// TwinCAT 3 PLC project CP_5C7432
// libraries:
//   AutomationBaseClasses, * (PTW TU Darmstadt)
//   Tc2_ControllerToolbox, * (Beckhoff Automation GmbH)
//   Tc2_Coupler, * (Beckhoff Automation GmbH)
//   Tc2_DALI, * (Beckhoff Automation GmbH)
//   Tc2_EIB, * (Beckhoff Automation GmbH)
//   Tc2_EtherCAT, * (Beckhoff Automation GmbH)
//   Tc2_IoFunctions, * (Beckhoff Automation GmbH)
//   Tc2_LON, * (Beckhoff Automation GmbH)
//   Tc2_MBus, * (Beckhoff Automation GmbH)
//   Tc2_ModbusRTU, * (Beckhoff Automation GmbH)
//   Tc2_ModbusSrv, * (Beckhoff Automation GmbH)
//   Tc2_Standard, * (Beckhoff Automation GmbH)
//   Tc2_Standard, * (Beckhoff Automation GmbH)
//   Tc2_System, * (Beckhoff Automation GmbH)
//   Tc2_System, * (Beckhoff Automation GmbH)
//   Tc2_SystemCX, * (Beckhoff Automation GmbH)
//   Tc2_Utilities, * (Beckhoff Automation GmbH)
//   Tc3_Module, * (Beckhoff Automation GmbH)
//   Tc3_Module, * (Beckhoff Automation GmbH)
//   Tc3_PLCopen_OpcUa, * (Beckhoff Automation GmbH)
// project tree:
//   DUTs/01 Actuators/pcmChiller/ E_PCMControlMode.TcDUT, ST_pcmChillerDefaultParameters.TcDUT, ST_pcmChillerState.TcDUT
//   DUTs/02 Sensors/ ST_JanitzaState.TcDUT
//   DUTs/03 Storages/BufferStorage/ ST_BufferStorageState.TcDUT
//   DUTs/03 Storages/HVFAStorage/ ST_HVFAStorageState.TcDUT (not stored), ST_HVFAStorageSystemDefaultParameters.TcDUT (not stored)
//   DUTs/03 Storages/PCMStorage/ ST_PCMStorageState.TcDUT
//   DUTs/03 Storages/VSIStorage/ ST_VSIStorageState.TcDUT (not stored), ST_VSIStorageSystemDefaultParameters.TcDUT (not stored)
//   DUTs/04 Systems/ConsumerSystems/CN/ ST_CN_CentralMachineCoolingDefaultParameters.TcDUT, ST_FlywheelMassStorageDefaultParameters.TcDUT
//   DUTs/04 Systems/ConsumerSystems/HNHT/ ST_AnnealingOvenExhaustGasDefaultParameters.TcDUT, ST_HNHT_CentralMachineHeatingDefaultParameters.TcDUT, ST_StaticHeatingDefaultParameters.TcDUT (not stored)
//   DUTs/04 Systems/ConsumerSystems/HNLT/ ST_AnnealingOvenSealingDefaultParameters.TcDUT (not stored), ST_DCSystemDefaultParameters.TcDUT, ST_CompressorDefaultParameters.TcDUT (not stored)
//   DUTs/04 Systems/CoolingSystems/AbsorptionChillerSystem/ ST_AbsorptionChillerDefaultParameters.TcDUT (not stored)
//   DUTs/04 Systems/CoolingSystems/eChiller/ ST_eChillerDefaultParameters.TcDUT, ST_eChillerState.TcDUT
//   DUTs/04 Systems/CoolingSystems/OuterCapillaryTubeMats/ ST_OuterCapillaryTubeMatsDefaultParameters.TcDUT (not stored)
//   DUTs/04 Systems/HeatingSystems/CHP/ E_CHPControlMode.TcDUT, ST_CHPDefaultParameters.TcDUT, ST_CHPSetParameters.TcDUT, ST_CHPState.TcDUT
//   DUTs/04 Systems/HeatingSystems/CondensingBoiler/ ST_CondensingBoilerDefaultParameters.TcDUT, ST_CondensingBoilerState.TcDUT
//   DUTs/04 Systems/HeatingSystems/HeatPump/ ST_HeatPumpDefaultParameters.TcDUT, ST_HeatPumpState.TcDUT
//   DUTs/04 Systems/LinkageSystems/HeatExchanger1/ ST_HeatExchanger1DefaultParameters.TcDUT
//   DUTs/04 Systems/LinkageSystems/InnerCapillaryTubeMats/ ST_InnerCapillaryTubeMatsDefaultParameters.TcDUT, ST_InnerCapillaryTubeMatsSetParameters.TcDUT (not stored)
//   DUTs/04 Systems/LinkageSystems/PCMSystem/ E_PCMSystemControlMode.TcDUT, ST_PCMSystemSetParameters.TcDUT
//   DUTs/04 Systems/LinkageSystems/UnderfloorHeating/ ST_UnderfloorHeatingDefaultParameters.TcDUT (not stored), ST_UnderfloorHeatingSetParameters.TcDUT (not stored)
//   DUTs/04 Systems/LinkageSystems/Ventilation/ ST_VentilationDefaultParameters.TcDUT, ST_VentilationSetParameters.TcDUT, ST_VentilationState.TcDUT
//   DUTs/04 Systems/StorageSystems/ ST_ActiveStorageSystemSetParameters.TcDUT (not stored), ST_ActiveStorageSystemState.TcDUT
//   DUTs/05 Thermal Networks/ ST_AmbientState.TcDUT, ST_CoolingNetworkControl.TcDUT, ST_HeatingNetworkHighTemperatureControl.TcDUT, ST_HnhtHnltLinkageControl.TcDUT, ST_HnltCnLinkageControl.TcDUT (not stored), ST_HeatingNetworkLowTemperatureControl.TcDUT (not stored), ST_HnhtCnLinkageControl.TcDUT, ST_ThermalNetworkState.TcDUT (not stored)
//   DUTs/06 Strategy/ ST_StrategyDefaultParameters.TcDUT, ST_StrategySetParameters.TcDUT, ST_StrategyState.TcDUT
//   DUTs/07 Utilities/ ST_OPC_UANode.TcDUT, ST_OPC_UA_Server.TcDUT (not stored)
//   DUTs/08 Lighting/Einzelanlagen/Beleuchtung %28Bel%29/ ST_Bel_Lampen_Monitoring.TcDUT (not stored), ST_Bel_Parameter.TcDUT (not stored), ST_Bel_RGBW_Steuerung.TcDUT (not stored), ST_Bel_RGBW_Zustand.TcDUT (not stored), ST_Bel_Stellwert.TcDUT (not stored), ST_Bel_Steuerung.TcDUT (not stored), ST_Bel_Zustand.TcDUT (not stored)
//   DUTs/08 Lighting/Einzelanlagen/RGBW-Kanal/ ST_RGBW_Steuerung.TcDUT (not stored), ST_RGBW_Zustand.TcDUT (not stored)
//   DUTs/08 Lighting/Library/Allgemein/ ST_Steuerung_auto_manu_BOOL.TcDUT (not stored), ST_Steuerung_auto_manu_opti_BOOL.TcDUT (not stored), ST_Steuerung_auto_manu_opti_REAL.TcDUT (not stored), ST_Steuerung_auto_manu_opti_SINT.TcDUT (not stored), ST_Steuerung_auto_manu_String.TcDUT (not stored), ST_Zustand_Netze_Anford.TcDUT (not stored), ST_Zustand_Netz_Anford.TcDUT (not stored)
//   DUTs/08 Lighting/Sonstige/ ST_GA_global.TcDUT (not stored), ST_Initialisierungsroutine.TcDUT (not stored)
//   DUTs/08 Lighting/Systeme/Beleuchtung %28Bel%29/ ST_System_Bel_Parameter.TcDUT (not stored), ST_System_Bel_Stellwert.TcDUT (not stored), ST_System_Bel_Steuerung.TcDUT (not stored), ST_System_Bel_Zustand.TcDUT (not stored)
//   GVLs/ GlobalVariables.TcGVL, M_Bus.TcGVL
//   GVLs/Lighting %28from old implementation%29/ Con_Bel.TcGVL (not stored), Global_Variables.TcGVL (not stored), Variablen_Konfiguration.TcGVL (not stored)
//   / MBus_WZaehler_Task.TcTTO, MBus_Zaehler_Task.TcTTO, Standard.TcTTO
//   POUs/01 Actuators/ConsumerUnits/ FB_AnnealingOven.TcPOU, FB_EMAG_GT.TcPOU, FB_DC.TcPOU, FB_EMAG_Y.TcPOU, FB_MAFAC_Java.TcPOU, FB_FlywheelMassStorage.TcPOU, FB_BvL_CleaningSystem.TcPOU, FB_Ventilation.TcPOU
//   POUs/01 Actuators/CoolingUnits/ FB_eChiller.TcPOU, FB_PCMChiller.TcPOU
//   POUs/01 Actuators/HeatingUnits/ FB_CHP.TcPOU, FB_HeatPump.TcPOU, FB_CondensingBoiler.TcPOU
//   POUs/01 Actuators/Pumps/ FB_Pump2Point.TcPOU
//   POUs/02 Sensors/ FB_JanitzaSensor.TcPOU, FB_LowVoltageMainDistribution.TcPOU, FB_WeatherStation.TcPOU
//   POUs/03 Storages/ FB_BufferStorage.TcPOU, FB_PCMStorage.TcPOU, FB_VSIStorage.TcPOU, FB_HVFAStorage.TcPOU
//   POUs/04 Systems/ConsumerSystems/CN/ FB_CN_CentralMachineCooling.TcPOU, FB_FlywheelMassStorageSystem.TcPOU
//   POUs/04 Systems/ConsumerSystems/HNHT/ FB_AnnealingOvenExhaustGasSystem.TcPOU, FB_HNHT_CentralMachineHeating.TcPOU, FB_StaticHeatingSystem.TcPOU
//   POUs/04 Systems/ConsumerSystems/HNLT/ FB_AnnealingOvenSealingSystem.TcPOU, FB_DCSystem.TcPOU, FB_CompressorSystem.TcPOU
//   POUs/04 Systems/CoolingSystems/ FB_AbsorptionChillerSystem.TcPOU, FB_eChillerSystem.TcPOU, FB_OuterCapillaryTubeMats.TcPOU, FB_PCMSupplySystem.TcPOU
//   POUs/04 Systems/HeatingSystems/ FB_CHPSystem.TcPOU, FB_CondensingBoilerSystem.TcPOU
//   POUs/04 Systems/LinkageSystems/ FB_HeatExchanger1System.TcPOU, FB_HeatPumpSystem_CN.TcPOU, FB_HeatPumpSystem_HNHT.TcPOU, FB_InnerCapillaryTubeMats.TcPOU, FB_UnderfloorHeatingSystem.TcPOU, FB_VentilationSystem.TcPOU
//   POUs/04 Systems/StorageSystems/ FB_HVFAStorageSystem.TcPOU, FB_VSIStorageSystem.TcPOU
//   POUs/05 Thermal Networks/ FB_Ambient.TcPOU, FB_CoolingNetwork.TcPOU, FB_HeatingNetworkHighTemperature.TcPOU, FB_HnhtCnLinkage.TcPOU, FB_HnhtHnltLinkage.TcPOU, FB_HnltCnLinkage.TcPOU, FB_HeatingNetworkLowTemperature.TcPOU
//   POUs/06 Strategy/ FB_StrategyController.TcPOU, FB_StrategyController_noChiller.TcPOU, FB_StrategyController_NoStorages.TcPOU, FB_StrategyController_Conventional.TcPOU
//   POUs/07 Utilities/ FB_OPC_UA_Read.TcPOU
//   POUs/08 Lighting/Einzelanlagen/Beleuchtung %28Bel%29/Bel_RGBW/ FB_Bel_Einzel_farbe.TcPOU (not stored), FB_Bel_Einzel_farbe_1.TcPOU (not stored), FB_Bel_RGBW.TcPOU (not stored), FB_Bel_RGBW_Ablaufsteuerung.TcPOU (not stored), FB_Bel_RGBW_Logik.TcPOU (not stored), FB_Bel_RGBW_Regelung.TcPOU (not stored), FB_Bel_RGBW_Sued.TcPOU (not stored) (excluded from build)
//   POUs/08 Lighting/Einzelanlagen/Beleuchtung %28Bel%29/ FB_Bel.TcPOU (not stored), FB_Bel_Ablaufsteuerung.TcPOU (not stored), FB_Bel_Filter.TcPOU (not stored), FB_Bel_Input.TcPOU (not stored), FB_Bel_Lichtsensor.TcPOU (not stored), FB_Bel_Logik.TcPOU (not stored), FB_Bel_Monitoring.TcPOU (not stored), FB_Bel_Output.TcPOU (not stored), FB_Bel_Sollwertscheck.TcPOU (not stored), FB_Bel_Stellwertscheck.TcPOU (not stored), FB_Bel_Steuerung.TcPOU (not stored), FB_Bel_Taster.TcPOU (not stored), FB_Bel_Taster_Steuerung.TcPOU (not stored), FB_Bel_Zustandscheck.TcPOU (not stored), F_Bel_Daten_Lesen.TcPOU (not stored), F_Bel_Daten_Schreiben.TcPOU (not stored)
//   POUs/08 Lighting/ FB_GA_Allgemein.TcPOU, FB_Initialisierungsroutine.TcPOU
//   POUs/08 Lighting/Library %28allgemein%29/ FB_SetResetFallTrigger.TcPOU (not stored)
//   POUs/08 Lighting/Systeme/Sonstiges/Beleuchtung/Beleuchtung Außen/ FB_System_BelAu.TcPOU (not stored), FB_System_BelAu_Ablaufsteuerung.TcPOU (not stored), FB_System_BelAu_Logik.TcPOU, FB_System_BelAu_Regelung.TcPOU, FB_System_BelAu_Sensorik.TcPOU, FB_System_BelAu_Sollwertscheck.TcPOU (not stored), FB_System_BelAu_Stellwertscheck.TcPOU (not stored), FB_System_BelAu_Zustandscheck.TcPOU (not stored)
//   POUs/08 Lighting/Systeme/Sonstiges/Beleuchtung/Beleuchtung Halle/ FB_System_BelHa.TcPOU (not stored), FB_System_BelHa_Ablaufsteuerung.TcPOU, FB_System_BelHa_Logik.TcPOU (not stored), FB_System_BelHa_Regelung.TcPOU (not stored), FB_System_BelHa_Sensorik.TcPOU, FB_System_BelHa_Sollwertscheck.TcPOU (not stored), FB_System_BelHa_Stellwertscheck.TcPOU, FB_System_BelHa_Zustandscheck.TcPOU
//   POUs/08 Lighting/Systeme/Sonstiges/Beleuchtung/ FB_Beleuchtung.TcPOU, FB_System_Bel_Zustandscheck.TcPOU (not stored)
//   POUs/ MAIN.TcPOU, MBUS_WZaehler.TcPOU, MBUS_WZaehler2.TcPOU, MBUS_WZaehler_Basement.TcPOU, MBUS_Zaehler.TcPOU
// real-time tasks:
//   TASK MBus_Zaehler_Task: cycle T#10ms, priority 8, ADS port 351
//   TASK Standard: cycle T#20ms, priority 10, ADS port 352
//   TASK MBus_WZaehler_Task: cycle T#6ms, priority 6, ADS port 353
//   TASK Gerät 7 (OPC UA Virtual)_Task_58: cycle T#40ms, priority 12, ADS port 350
// I/O:
//   DEVICE Gerät 6 (EL6731), AmsNetId 0.0.0.0.7.1
//     Box 1 (CIM/CIU 150 pump) // Vendor: GRUNDFOS Revision: R1 PU361
//     Box 2 (CIM/CIU 150 pump) // Vendor: GRUNDFOS Revision: R1 PU261
//     Box 3 (CIM/CIU 150 pump) // Vendor: GRUNDFOS Revision: R1 PU300
//     Box 4 (CIM/CIU 150 pump) // Vendor: GRUNDFOS Revision: R1 PU100
//     Box 5 (CIM/CIU 150 pump) // Vendor: GRUNDFOS Revision: R1 PU145
//     Box 6 (CIM/CIU 150 pump) // Vendor: GRUNDFOS Revision: R1 PU245
//   DEVICE Gerät 10 (EtherCAT), AmsNetId 0.0.0.0.11.1
//     Term 31 (EK1100) [EK1100 EtherCAT Coupler (2A E-Bus)]
//       Term 30 (EL6070-0033) [EL6070-0033 1Ch. Licence key terminal, individual licences]
//       Profibus_1 (EL6731) [EL6731 PROFIBUS DP Master]
//       Profibus_2 (EL6731) [EL6731 PROFIBUS DP Master]
//       Box 3 (BK1250)
//     Klemme 15 (EK1100) [EK1100 EtherCAT-Koppler (2A E-Bus)]
//       Klemme 27 (EL3068) [EL3068 8K. Ana. Eingang 0-10V]
//       Klemme 28 (EL4008) [EL4008 8K. Ana. Ausgang 0-10V, 12bit]
//       Klemme 39 (EK1521-0010) [EK1521-0010 1-Port EtherCAT-Abzweig (FX-SingleMode)]
//         Klemme 40 (EK1501-0010) [EK1501-0010 EtherCAT-Koppler (2A E-Bus, FX-SingleMode, ID-Switch)]
//           Klemme 41 (EL2809) [EL2809 16K. Dig. Ausgang 24V, 0.5A]
//           Klemme 42 (EL4008) [EL4008 8K. Ana. Ausgang 0-10V, 12bit]
//           Klemme 43 (EL1809) [EL1809 16K. Dig. Eingang 24V, 3ms]
//           Klemme 51 (EL3068) [EL3068 8K. Ana. Eingang 0-10V]
//           Klemme 53 (EL4008) [EL4008 8K. Ana. Ausgang 0-10V, 12bit]
//           Klemme 78 (EL3202-0010) [EL3202-0010 2K. Ana. Eingang PT100 (RTD), hochgenau]
//           Klemme 79 (EL3202-0010) [EL3202-0010 2K. Ana. Eingang PT100 (RTD), hochgenau]
//           Klemme 80 (EL3202-0010) [EL3202-0010 2K. Ana. Eingang PT100 (RTD), hochgenau]
//           Klemme 81 (EL3202-0010) [EL3202-0010 2K. Ana. Eingang PT100 (RTD), hochgenau]
//           Klemme 23 (EL6731) [EL6731 PROFIBUS DP Master]
//           Box 36 (BK1250)
//       Klemme 25 (EL9011) [EL9011 Endklemme]
//       Box 4 (BK1250)
//     Klemme 64 (EK1100) [EK1100 EtherCAT-Koppler (2A E-Bus)]
//       Klemme 65 (EL3202-0010) [EL3202-0010 2K. Ana. Eingang PT100 (RTD), hochgenau]
//       Klemme 66 (EL3202-0010) [EL3202-0010 2K. Ana. Eingang PT100 (RTD), hochgenau]
//       Klemme 67 (EL3068) [EL3068 8K. Ana. Eingang 0-10V]
//       Klemme 68 (EL4008) [EL4008 8K. Ana. Ausgang 0-10V, 12bit]
//       Klemme 69 (EL1809) [EL1809 16K. Dig. Eingang 24V, 3ms]
//       Klemme 70 (EL2809) [EL2809 16K. Dig. Ausgang 24V, 0.5A]
//       Klemme 87 (EL3218) [EL3218-0000 8K. Ana. Eingang PT100 (RTD)]
//       Klemme 88 (EL4002) [EL4002 2K. Ana. Ausgang 0-10V, 12bit]
//       Klemme 89 (EL3062-0030) [EL3062-0030 2K.Ana. Eingang 0-30V]
//       Box 55 (BK1250)
//   DEVICE Device 2 (EL6731), AmsNetId 0.0.0.0.3.1
//     Box 1 (CIM/CIU 150 pump) // Vendor: GRUNDFOS Revision: R1 PU235
//     Box 3 (CIM/CIU 150 pump) // Vendor: GRUNDFOS Revision: R1 PU215
//     Box 4 (CIM/CIU 150 pump) // Vendor: GRUNDFOS Revision: R1 PU315
//     Box 5 (CIM/CIU 150 pump) // Vendor: GRUNDFOS Revision: R1 PU322
//     Box 6 (CIM/CIU 150 pump) // Vendor: GRUNDFOS Revision: R1 PU321
//     Box 9 (CIM/CIU 150 pump) // Vendor: GRUNDFOS Revision: R1 PU600
//     Box 10 (CIM/CIU 150 pump) // Vendor: GRUNDFOS Revision: R1 PU500
//     Box 11 (CIM/CIU 150 pump) // Vendor: GRUNDFOS Revision: R1 PU425
//     Box 13 (CIM/CIU 150 pump) // Vendor: GRUNDFOS Revision: R1 PU405
//     Box 14 (CIM/CIU 150 pump) // Vendor: GRUNDFOS Revision: R1 PU251
//     Box 15 (CIM/CIU 150 pump) // Vendor: GRUNDFOS Revision: R1 PU455
//     Box 16 (CIM/CIU 150 pump) // Vendor: GRUNDFOS Revision: R1 PU350
//     Box 17 (CIM/CIU 150 pump) (disabled) // Vendor: GRUNDFOS Revision: R1 PU191
//     Box 18 (GSD Box) (Mkv Gateway) (disabled) // Vendor: AtlasCopco Revision: 0.00
//     Box 19 (GSD Box) (UMG604) (disabled) // Vendor: Janitza electronics GmbH Revision: Rev. 1
//     Box 20 (CIM/CIU 150 pump) // Vendor: GRUNDFOS Revision: R1 PU305
//     Box 21 (CIM/CIU 150 pump) // Vendor: GRUNDFOS Revision: R1 PU306
//     Box 22 (CIM/CIU 150 pump) // Vendor: GRUNDFOS Revision: R1 PU242
//   DEVICE Gerät 1 (EL6731), AmsNetId 0.0.0.0.2.1
//     Box 1 (CIM/CIU 150 pump) // Vendor: GRUNDFOS Revision: R1 PU205
//     Box 2 (CIM/CIU 150 pump) // Vendor: GRUNDFOS Revision: R1 PU105
//   DEVICE Gerät 7 (OPC UA Virtual), AmsNetId 0.0.0.0.8.1
//   DEVICE Device 8 (EtherCAT), AmsNetId 0.0.0.0.9.1
//     Term 36 (EK1100) [EK1100 EtherCAT Coupler (2A E-Bus)]
//       Term 37 (EL2008) [EL2008 8Ch. Dig. Output 24V, 0.5A]
//       Term 38 (EL1008) [EL1008 8Ch. Dig. Input 24V, 3ms]
//       Term 45 (EL4004) [EL4004 4Ch. Ana. Output 0-10V, 12bit]
//       Term 47 (EL3008) [EL3008 8Ch. Ana. Input +/-10V]
//       Term 48 (EL3152) [EL3152 2Ch. Ana Input 4-20mA]
//       Term 49 (EL3152) [EL3152 2Ch. Ana Input 4-20mA]
//       Term 50 (EL3008) [EL3008 8Ch. Ana. Input +/-10V]
//       Term 52 (EL3218) [EL3218-0000 8Ch. Ana. Input PT100 (RTD)]
//       Term 10 (EL9011) [EL9011 End Terminal]
// variable links:
//   CP_5C7432/CP_5C7432 Instance <-> Device 1 (EL6731)/Box 1 (CIM/CIU 150 pump)
//     Standard Inputs/MAIN.HNLT.HVFASystem.PUx05.StatusModule_IN <-> StatusModule/Inputs/StatusModule_0_0
//     Standard Inputs/MAIN.HNLT.HVFASystem.PUx05.fActualSetpoint_IN <-> ActualSetpoint/Inputs/ActualSetpoint_0_0
//     Standard Inputs/MAIN.HNLT.HVFASystem.PUx05.fPowerElectric_IN <-> Power/Inputs/Power_0_0
//     Standard Inputs/MAIN.HNLT.HVFASystem.PUx05.fPowerThermal_IN <-> HeatPower/Inputs/HeatPower_0_0
//     Standard Inputs/MAIN.HNLT.HVFASystem.PUx05.fPressureDifference_IN <-> DiffPressure/Inputs/DiffPressure_0_0
//     Standard Inputs/MAIN.HNLT.HVFASystem.PUx05.fRotationalSpeed_IN <-> Speed/Inputs/Speed_0_0
//     Standard Inputs/MAIN.HNLT.HVFASystem.PUx05.fTemperatureDifference_IN <-> HeatDiffTemp/Inputs/HeatDiffTemp_0_0
//     Standard Inputs/MAIN.HNLT.HVFASystem.PUx05.fTemperatureExternal_IN <-> RemoteTemp2/Inputs/RemoteTemp2_0_0
//     Standard Inputs/MAIN.HNLT.HVFASystem.PUx05.fVolumeFlowRate_IN <-> VolumeFlow/Inputs/VolumeFlow_0_0
//     Standard Inputs/MAIN.HNLT.HVFASystem.PUx05.nAlarmCode_IN <-> FaultCode/Inputs/FaultCode_0_0
//     Standard Inputs/MAIN.HNLT.HVFASystem.PUx05.nWarningCode_IN <-> WarningCode/Inputs/WarningCode_0_0
//     Standard Inputs/MAIN.HNLT.HVFASystem.PUx05.stTemperatureInternal_Genibus_Reply <-> DirectDataReply/Inputs/DirectDataReply_0_0
//     Standard Outputs/MAIN.HNLT.HVFASystem.PUx05.ControlModule_OUT <-> ControlModule/Outputs/ControlModule_1_0
//     Standard Outputs/MAIN.HNLT.HVFASystem.PUx05.stTemperatureInternal_Genibus_Request <-> DirectDataRequest/Outputs/DirectDataRequest_1_0
//   CP_5C7432/CP_5C7432 Instance <-> Device 1 (EL6731)/Box 2 (CIM/CIU 150 pump)
//     Standard Inputs/MAIN.CN.HVFASystem.PUx05.StatusModule_IN <-> StatusModule/Inputs/StatusModule_0_0
//     Standard Inputs/MAIN.CN.HVFASystem.PUx05.fActualSetpoint_IN <-> ActualSetpoint/Inputs/ActualSetpoint_0_0
//     Standard Inputs/MAIN.CN.HVFASystem.PUx05.fPowerElectric_IN <-> Power/Inputs/Power_0_0
//     Standard Inputs/MAIN.CN.HVFASystem.PUx05.fPowerThermal_IN <-> HeatPower/Inputs/HeatPower_0_0
//     Standard Inputs/MAIN.CN.HVFASystem.PUx05.fPressureDifference_IN <-> DiffPressure/Inputs/DiffPressure_0_0
//     Standard Inputs/MAIN.CN.HVFASystem.PUx05.fRotationalSpeed_IN <-> Speed/Inputs/Speed_0_0
//     Standard Inputs/MAIN.CN.HVFASystem.PUx05.fTemperatureDifference_IN <-> HeatDiffTemp/Inputs/HeatDiffTemp_0_0
//     Standard Inputs/MAIN.CN.HVFASystem.PUx05.fTemperatureExternal_IN <-> RemoteTemp2/Inputs/RemoteTemp2_0_0
//     Standard Inputs/MAIN.CN.HVFASystem.PUx05.fVolumeFlowRate_IN <-> VolumeFlow/Inputs/VolumeFlow_0_0
//     Standard Inputs/MAIN.CN.HVFASystem.PUx05.nAlarmCode_IN <-> FaultCode/Inputs/FaultCode_0_0
//     Standard Inputs/MAIN.CN.HVFASystem.PUx05.nWarningCode_IN <-> WarningCode/Inputs/WarningCode_0_0
//     Standard Inputs/MAIN.CN.HVFASystem.PUx05.stTemperatureInternal_Genibus_Reply <-> DirectDataReply/Inputs/DirectDataReply_0_0
//     Standard Outputs/MAIN.CN.HVFASystem.PUx05.ControlModule_OUT <-> ControlModule/Outputs/ControlModule_1_0
//     Standard Outputs/MAIN.CN.HVFASystem.PUx05.stTemperatureInternal_Genibus_Request <-> DirectDataRequest/Outputs/DirectDataRequest_1_0
//   CP_5C7432/CP_5C7432 Instance <-> Device 10 (EtherCAT)/Term 15 (EK1100)/Box 4 (BK1250)
//     MBus_WZaehler_Task Inputs/.IN_WZaehler/D <-> Term 48 (KL6781)/Channel 1/Data In 0
//     MBus_WZaehler_Task Inputs/.IN_WZaehler/D @bit {8..168 step 8} <-> Term 48 (KL6781)/Channel 1/Data In {1..21}  (21 links)
//     MBus_WZaehler_Task Inputs/.IN_WZaehler/Status <-> Term 48 (KL6781)/Channel 1/State
//     MBus_WZaehler_Task Outputs/.OUT_WZaehler/Ctrl <-> Term 48 (KL6781)/Channel 1/Ctrl
//     MBus_WZaehler_Task Outputs/.OUT_WZaehler/D <-> Term 48 (KL6781)/Channel 1/Data Out 0
//     MBus_WZaehler_Task Outputs/.OUT_WZaehler/D @bit {8..168 step 8} <-> Term 48 (KL6781)/Channel 1/Data Out {1..21}  (21 links)
//   CP_5C7432/CP_5C7432 Instance <-> Device 10 (EtherCAT)/Term 15 (EK1100)/Term 27 (EL3068)
//     Standard Inputs/MAIN.HNHT.AnnealingOvenExhaustGasSystem.RV361.nOperatingPoint_IN <-> ai_RV361/ai_RV361
//     Standard Inputs/MAIN.HNHT.CHP1System.RV32x.nOperatingPoint_IN <-> ai_RV321/ai_RV321
//     Standard Inputs/MAIN.HNHT.CHP2System.RV32x.nOperatingPoint_IN <-> ai_RV322/ai_RV322
//     Standard Inputs/MAIN.HNHT.CondensingBoilerSystem.RV331.nOperatingPoint_IN <-> ai_RV331/ai_RV331
//     Standard Inputs/MAIN.HNHT_HNLT.HeatExchanger1System.RV315.nOperatingPoint_IN <-> ai_RV315/ai_RV315
//     Standard Inputs/MAIN.HNLT.AnnealingOvenSealingSystem.RV261.nOperatingPoint_IN <-> ai_RV261/ai_RV261
//     Standard Inputs/MAIN.HNLT.CompressorSystem.RV251.nOperatingPoint_IN <-> ai_RV251/ai_RV251
//   CP_5C7432/CP_5C7432 Instance <-> Device 10 (EtherCAT)/Term 15 (EK1100)/Term 28 (EL4008)
//     Standard Outputs/MAIN.HNHT.AnnealingOvenExhaustGasSystem.RV361.nSetPoint_OUT <-> ao_RV361/ao_RV361
//     Standard Outputs/MAIN.HNHT.CHP1System.RV32x.nSetPoint_OUT <-> ao_RV321/ao_RV321
//     Standard Outputs/MAIN.HNHT.CHP2System.RV32x.nSetPoint_OUT <-> ao_RV322/ao_RV322
//     Standard Outputs/MAIN.HNHT.CondensingBoilerSystem.RV331.nSetPoint_OUT <-> ao_RV331/ao_RV331
//     Standard Outputs/MAIN.HNHT_HNLT.HeatExchanger1System.RV315.nSetPoint_OUT <-> ao_RV315/ao_RV315
//     Standard Outputs/MAIN.HNLT.AnnealingOvenSealingSystem.RV261.nSetPoint_OUT <-> ao_RV261/ao_RV261
//     Standard Outputs/MAIN.HNLT.CompressorSystem.RV251.nSetPoint_OUT <-> ao_RV251/ao_RV251
//   CP_5C7432/CP_5C7432 Instance <-> Device 10 (EtherCAT)/Term 15 (EK1100)/Term 39 (EK1521-0010)/Term 40 (EK1501-0010)/Box 36 (BK1250)
//     MBus_WZaehler_Task Inputs/.IN_WZaehler2/D <-> Term 98 (KL6781)/Channel 1/Data In 0
//     MBus_WZaehler_Task Inputs/.IN_WZaehler2/D @bit {8..168 step 8} <-> Term 98 (KL6781)/Channel 1/Data In {1..21}  (21 links)
//     MBus_WZaehler_Task Inputs/.IN_WZaehler2/Status <-> Term 98 (KL6781)/Channel 1/Status
//     MBus_WZaehler_Task Outputs/.OUT_WZaehler2/Ctrl <-> Term 98 (KL6781)/Channel 1/Ctrl
//     MBus_WZaehler_Task Outputs/.OUT_WZaehler2/D <-> Term 98 (KL6781)/Channel 1/Data Out 0
//     MBus_WZaehler_Task Outputs/.OUT_WZaehler2/D @bit {8..168 step 8} <-> Term 98 (KL6781)/Channel 1/Data Out {1..21}  (21 links)
//     Standard Inputs/MAIN.Ambient.AmbientTemperatureSensor_Container.temperature_IN <-> Term 100 (KL3214)/Channel 1/Daten Ein
//   CP_5C7432/CP_5C7432 Instance <-> Device 10 (EtherCAT)/Term 15 (EK1100)/Term 39 (EK1521-0010)/Term 40 (EK1501-0010)/Term 41 (EL2809)
//     Standard Outputs/MAIN.CN.HVFASystem.PU7x0.bSetStatusOn_OUT <-> bo_PU710/bo_PU710
//     Standard Outputs/MAIN.CN.eChillerSystem.eChiller.bSetStatusOn_OUT <-> bo_eChiller/bo_eChiller
//     Standard Outputs/MAIN.HNLT.HVFASystem.PU7x0.bSetStatusOn_OUT <-> bo_PU720/bo_PU720
//   CP_5C7432/CP_5C7432 Instance <-> Device 10 (EtherCAT)/Term 15 (EK1100)/Term 39 (EK1521-0010)/Term 40 (EK1501-0010)/Term 42 (EL4008)
//     Standard Outputs/MAIN.CN.HVFASystem.RVx05.nSetPoint_OUT <-> ao_RV105/ao_RV105
//     Standard Outputs/MAIN.CN.HVFASystem.SVx05.nSetPoint_OUT <-> ao_SV105/ao_SV105
//     Standard Outputs/MAIN.CN.HVFASystem.SVx06.nSetPoint_OUT <-> ao_SV106/ao_SV106
//     Standard Outputs/MAIN.CN.eChillerSystem.SV138.nSetPoint_OUT <-> ao_SV138/ao_SV138
//     Standard Outputs/MAIN.HNLT.HVFASystem.RVx05.nSetPoint_OUT <-> ao_RV205/ao_RV205
//     Standard Outputs/MAIN.HNLT.HVFASystem.SVx05.nSetPoint_OUT <-> ao_SV205/ao_SV205
//     Standard Outputs/MAIN.HNLT.HVFASystem.SVx06.nSetPoint_OUT <-> ao_SV206/ao_SV206
//   CP_5C7432/CP_5C7432 Instance <-> Device 10 (EtherCAT)/Term 15 (EK1100)/Term 39 (EK1521-0010)/Term 40 (EK1501-0010)/Term 43 (EL1809)
//     Standard Inputs/MAIN.CN.eChillerSystem.eChiller.bError_IN <-> bi_eChiller_bError/bi_eChiller_bError
//     Standard Inputs/MAIN.CN.eChillerSystem.eChiller.bStatusOn_IN <-> bi_eChiller_bStatusOn/bi_eChiller_bStatusOn
//     Standard Inputs/MAIN.CN.eChillerSystem.eChiller.bWarning_IN <-> bi_eChiller_bWarning/bi_eChiller_bWarning
//   CP_5C7432/CP_5C7432 Instance <-> Device 10 (EtherCAT)/Term 15 (EK1100)/Term 39 (EK1521-0010)/Term 40 (EK1501-0010)/Term 51 (EL3068)
//     Standard Inputs/MAIN.CN.HVFASystem.RVx05.nOperatingPoint_IN <-> ai_RV105/ai_RV105
//     Standard Inputs/MAIN.CN.HVFASystem.SVx05.nOperatingPoint_IN <-> ai_SV105/ai_SV105
//     Standard Inputs/MAIN.CN.HVFASystem.SVx06.nOperatingPoint_IN <-> ai_SV106/ai_SV106
//     Standard Inputs/MAIN.CN.eChillerSystem.SV138.nOperatingPoint_IN <-> ai_SV138/ai_SV138
//     Standard Inputs/MAIN.HNLT.HVFASystem.RVx05.nOperatingPoint_IN <-> ai_RV205/ai_RV205
//     Standard Inputs/MAIN.HNLT.HVFASystem.SVx05.nOperatingPoint_IN <-> ai_SV205/ai_SV205
//     Standard Inputs/MAIN.HNLT.HVFASystem.SVx06.nOperatingPoint_IN <-> ai_SV206/ai_SV206
//   CP_5C7432/CP_5C7432 Instance <-> Device 10 (EtherCAT)/Term 15 (EK1100)/Term 39 (EK1521-0010)/Term 40 (EK1501-0010)/Term 53 (EL4008)
//     Standard Outputs/MAIN.CN.eChillerSystem.eChiller.nActualTemperature_OUT <-> ao_eChiller_ActualTemperature_BufferStorage/ao_eChiller_ActualTemperature_BufferStorage
//     Standard Outputs/MAIN.CN.eChillerSystem.eChiller.nReturnTemperature_Consumers_OUT <-> ao_eChiller_ReturnTemperature_Consumers/ao_eChiller_ReturnTemperature_Consumers
//     Standard Outputs/MAIN.CN.eChillerSystem.eChiller.nSetPoint_OUT <-> ao_eChiller_fSetPoint/ao_eChiller_fSetPoint
//   CP_5C7432/CP_5C7432 Instance <-> Device 10 (EtherCAT)/Term 15 (EK1100)/Term 39 (EK1521-0010)/Term 40 (EK1501-0010)/Term 78 (EL3202-0010)
//     Standard Inputs/MAIN.HNLT.HVFASystem.HVFAStorage.LowerTemperatureSensor.temperature_IN <-> TF797_HNLT_HVFA_LowerTemperature/TF797_HNLT_HVFA_LowerTemperature
//     Standard Inputs/MAIN.HNLT.HVFASystem.HVFAStorage.UpperTemperatureSensor.temperature_IN <-> TF797_HNLT_HVFA_UpperTemperature/TF797_HNLT_HVFA_UpperTemperature
//   CP_5C7432/CP_5C7432 Instance <-> Device 10 (EtherCAT)/Term 15 (EK1100)/Term 39 (EK1521-0010)/Term 40 (EK1501-0010)/Term 79 (EL3202-0010)
//     Standard Inputs/MAIN.CN.HVFASystem.HVFAStorage.LowerTemperatureSensor.temperature_IN <-> TF796_CN_HVFA_LowerTemperature/TF796_CN_HVFA_LowerTemperature
//   CP_5C7432/CP_5C7432 Instance <-> Device 10 (EtherCAT)/Term 15 (EK1100)/Term 39 (EK1521-0010)/Term 40 (EK1501-0010)/Term 80 (EL3202-0010)
//     Standard Inputs/MAIN.CN.HVFASystem.HVFAStorage.UpperTemperatureSensor.temperature_IN <-> TF795_CN_HVFA_UpperTemperature/TF795_CN_HVFA_UpperTemperature
//   CP_5C7432/CP_5C7432 Instance <-> Device 10 (EtherCAT)/Term 15 (EK1100)/Term 39 (EK1521-0010)/Term 40 (EK1501-0010)/Term 81 (EL3202-0010)
//     Standard Inputs/MAIN.Ambient.RoomTemperatureSensor_Container.temperature_IN <-> TF061_RoomTemperature_Container/TF061_RoomTemperature_Container
//   CP_5C7432/CP_5C7432 Instance <-> Device 10 (EtherCAT)/Term 31 (EK1100)/Box 3 (BK1250)
//     MBus_Zaehler_Task Inputs/.IN_Stromzaehler/D[{0..21}] <-> K525A1_M_Bus/Channel 1/Data In {0..21}  (22 links)
//     MBus_Zaehler_Task Inputs/.IN_Stromzaehler/Status <-> K525A1_M_Bus/Channel 1/Status
//     MBus_Zaehler_Task Outputs/.OUT_Stromzaehler/Ctrl <-> K525A1_M_Bus/Channel 1/Ctrl
//     MBus_Zaehler_Task Outputs/.OUT_Stromzaehler/D[{0..21}] <-> K525A1_M_Bus/Channel 1/Data Out {0..21}  (22 links)
//     Standard Inputs/.Beleuchtung.Hallenbeleuchtung.Sensor1.IN_Helligkeit <-> K560A1_AI-2/2/ai_Lichtsensor_Halle_Gruppe_01/ai_Lichtsensor_Halle_Gruppe_01
//     Standard Inputs/.Beleuchtung.Hallenbeleuchtung.Sensor2.IN_Helligkeit <-> K560A1_AI-2/2/ai_Lichtsensor_Halle_Gruppe_02/ai_Lichtsensor_Halle_Gruppe_02
//     Standard Inputs/.Beleuchtung.Hallenbeleuchtung.Steuer_Taster.IN_Bin <-> K581A1_BI (KL1408)/LI000_Licht_Halle_Gruppe_02_Taster/LI000_Licht_Halle_Gruppe_02_Taster
//     Standard Inputs/.Beleuchtung.Hallenbeleuchtung.TasterGruppe1.IN_Bin <-> K581A1_BI (KL1408)/LI000_Licht_Halle_Gruppe_01_Taster/LI000_Licht_Halle_Gruppe_01_Taster
//     Standard Inputs/.Dali_K522A1_DALI_IN/nData <-> K522A1_DALI/Channel 1/Daten Ein
//     Standard Inputs/.Dali_K522A1_DALI_IN/nStatus <-> K522A1_DALI/Channel 1/Status
//     Standard Inputs/MAIN.Ambient.HallTemperatureSensor_Section1.temperature_IN <-> K578A1_AI (KL3222)/TF051_HallTemperature_Section1/TF051_HallTemperature_Section1
//     Standard Inputs/MAIN.Ambient.HallTemperatureSensor_Section2.temperature_IN <-> K579A1_AI (KL3222)/TF052_HallTemperature_Section2/TF052_HallTemperature_Section2
//     Standard Inputs/MAIN.Ambient.HallTemperatureSensor_Section3.temperature_IN <-> K579A1_AI (KL3222)/TF053_HallTemperature_Section3/TF053_HallTemperature_Section3
//     Standard Inputs/MAIN.Ambient.WeatherStation.KL6301_IN @bit {16..184 step 8} <-> K523A1_EIB/Channel 1/Input Data {1..22}  (22 links)
//     Standard Inputs/MAIN.Ambient.WeatherStation.KL6301_IN <-> K523A1_EIB/Channel 1/Parameter Status
//     Standard Inputs/MAIN.CN.BufferStorage.LowerTemperatureSensor.temperature_IN <-> K550A1_AI-2/2/ai_TF195_CN_LowerTemperature/ai_TF195_CN_LowerTemperature
//     Standard Inputs/MAIN.CN.BufferStorage.MidTemperatureSensor.temperature_IN <-> K550A1_AI-2/2/ai_TF195_CN_MidTemperature/ai_TF195_CN_MidTemperature
//     Standard Inputs/MAIN.CN.BufferStorage.PressureSensor.nPressure_IN <-> K560A1_AI-1/2/ai_PS100/ai_PS100
//     Standard Inputs/MAIN.CN.BufferStorage.UpperTemperatureSensor.temperature_IN <-> K550A1_AI-2/2/ai_TF195_CN_UpperTemperature/ai_TF195_CN_UpperTemperature
//     Standard Inputs/MAIN.CN.CentralMachineCoolingSystem.SV100.bStatusOff_IN <-> K531A1_BI/bi_SV100_Closed/bi_SV100_Closed
//     Standard Inputs/MAIN.CN.CentralMachineCoolingSystem.SV100.bStatusOn_IN <-> K531A1_BI/bi_SV100_Open/bi_SV100_Open
//     Standard Inputs/MAIN.HNHT.BufferStorage.PressureSensor.nPressure_IN <-> K560A1_AI-1/2/ai_PS300/ai_PS300
//     Standard Inputs/MAIN.HNHT.CHP1System.CHP.bError_IN <-> K531A1_BI/bi_CHP1_Error/bi_CHP1_Error
//     Standard Inputs/MAIN.HNHT.CHP2System.CHP.bError_IN <-> K535A1_BI/bi_CHP2_Error/bi_CHP2_Error
//     Standard Inputs/MAIN.HNHT.CHP1System.SV32x.bStatusOff_IN <-> K533A1_BI/bi_SV321_Closed/bi_SV321_Closed
//     Standard Inputs/MAIN.HNHT.CHP2System.SV32x.bStatusOff_IN <-> K531A1_BI/bi_SV322_Closed/bi_SV322_Closed
//     Standard Inputs/MAIN.HNHT.CHP1System.SV32x.bStatusOn_IN <-> K533A1_BI/bi_SV321_Open/bi_SV321_Open
//     Standard Inputs/MAIN.HNHT.CHP2System.SV32x.bStatusOn_IN <-> K533A1_BI/bi_SV322_Open/bi_SV322_Open
//     Standard Inputs/MAIN.HNHT.CondensingBoilerSystem.SV331.bStatusOff_IN <-> K531A1_BI/bi_SV331_Closed/bi_SV331_Closed
//     Standard Inputs/MAIN.HNHT.CondensingBoilerSystem.SV331.bStatusOn_IN <-> K533A1_BI/bi_SV331_Open/bi_SV331_Open
//     Standard Inputs/MAIN.HNHT.VSIStorageSystem.VSIStorage.LowerTemperatureSensor.temperature_IN <-> K578A1_AI (KL3222)/TF395_VSI _LowerTemperature/TF395_VSI _LowerTemperature
//     Standard Inputs/MAIN.HNHT.VSIStorageSystem.VSIStorage.MidTemperatureSensor.temperature_IN <-> K577A1_AI (KL3222)/TF395_VSI _MidTemperature/TF395_VSI _MidTemperature
//     Standard Inputs/MAIN.HNHT.VSIStorageSystem.VSIStorage.UpperTemperatureSensor.temperature_IN <-> K577A1_AI (KL3222)/TF395_VSI _UpperTemperature/TF395_VSI _UpperTemperature
//     Standard Inputs/MAIN.HNHT_CN.VentilationSystem.SV453.bStatusOff_IN <-> K535A1_BI/bi_SV453_Closed/bi_SV453_Closed
//     Standard Inputs/MAIN.HNHT_CN.VentilationSystem.SV454.bStatusOff_IN <-> K535A1_BI/bi_SV454_Closed/bi_SV454_Closed
//     Standard Inputs/MAIN.HNHT_CN.VentilationSystem.SV453.bStatusOn_IN <-> K535A1_BI/bi_SV453_Open/bi_SV453_Open
//     Standard Inputs/MAIN.HNHT_CN.VentilationSystem.SV454.bStatusOn_IN <-> K535A1_BI/bi_SV454_Open/bi_SV454_Open
//     Standard Inputs/MAIN.HNLT.BufferStorage.LowerTemperatureSensor.temperature_IN <-> K550A1_AI-1/2/ai_TF295_HNLT_LowerTemperature/ai_TF295_LowerTemperature
//     Standard Inputs/MAIN.HNLT.BufferStorage.MidTemperatureSensor.temperature_IN <-> K550A1_AI-1/2/ai_TF295_HNLT_MidTemperature/ai_TF295_MidTemperature
//     Standard Inputs/MAIN.HNLT.BufferStorage.PressureSensor.nPressure_IN <-> K560A1_AI-1/2/ai_PS200/ai_PS200
//     Standard Inputs/MAIN.HNLT.BufferStorage.UpperTemperatureSensor.temperature_IN <-> K550A1_AI-2/2/ai_TF295_HNLT_UpperTemperature/ai_TF295_HNLT_UpperTemperature
//     Standard Inputs/MAIN.HNLT.OuterCapillaryTubeMats.PS600.nPressure_IN <-> K560A1_AI-2/2/ai_PS600/ai_PS600
//     Standard Inputs/MAIN.HNLT.OuterCapillaryTubeMats.SV605.bStatusOff_IN <-> K535A1_BI/bi_SV605_Closed/bi_SV605_closed
//     Standard Inputs/MAIN.HNLT.OuterCapillaryTubeMats.SV605.bStatusOn_IN <-> K535A1_BI/bi_SV605_Open/bi_SV605_open
//     Standard Inputs/MAIN.HNLT.OuterCapillaryTubeMats.TS640.temperature_IN <-> K553A1_AI-2/2/ai_TF640/ai_TF640
//     Standard Inputs/MAIN.HNLT.OuterCapillaryTubeMats.TS660.temperature_IN <-> K553A1_AI-2/2/ai_TF660/ai_TF660
//     Standard Inputs/MAIN.HNLT_CN.InnerCapillaryTubeMats.PS500.nPressure_IN <-> K560A1_AI-1/2/ai_DS500/ai_PS500
//     Standard Inputs/MAIN.HNLT_CN.InnerCapillaryTubeMats.SV505.bStatusOff_IN <-> K533A1_BI/bi_SV505_Closed/bi_SV505_Closed
//     Standard Inputs/MAIN.HNLT_CN.InnerCapillaryTubeMats.SV505.bStatusOn_IN <-> K533A1_BI/bi_SV505_Open/bi_SV505_Open
//     Standard Inputs/MAIN.HNLT_CN.InnerCapillaryTubeMats.SV_CN.bStatusOff_IN <-> K533A1_BI/bi_SV_CN_HeatExchanger3_Closed/bi_SV_CN_HeatExchanger3_Closed
//     Standard Inputs/MAIN.HNLT_CN.InnerCapillaryTubeMats.SV_CN.bStatusOn_IN <-> K533A1_BI/bi_SV_CN_HeatExchanger3_Open/bi_SV_CN_HeatExchanger3_Open
//     Standard Inputs/MAIN.HNLT_CN.InnerCapillaryTubeMats.SV_HNLT.bStatusOff_IN <-> K533A1_BI/bi_SV_HNLT_HeatExchanger3_Closed/bi_SV_HNLT_HeatExchanger3_Closed
//     Standard Inputs/MAIN.HNLT_CN.InnerCapillaryTubeMats.SV_HNLT.bStatusOn_IN <-> K533A1_BI/bi_SV_HNLT_HeatExchanger3_Open/bi_SV_HNLT_HeatExchanger3_Open
//     Standard Inputs/MAIN.HNLT_CN.InnerCapillaryTubeMats.TS541.temperature_IN <-> K552A1_AI-1/2/ai_TF541/ai_TF541
//     Standard Inputs/MAIN.HNLT_CN.InnerCapillaryTubeMats.TS542.temperature_IN <-> K552A1_AI-1/2/ai_TF542/ai_TF542
//     Standard Inputs/MAIN.HNLT_CN.InnerCapillaryTubeMats.TS543.temperature_IN <-> K552A1_AI-1/2/ai_TF543/ai_TF543
//     Standard Inputs/MAIN.HNLT_CN.InnerCapillaryTubeMats.TS551.temperature_IN <-> K552A1_AI-1/2/ai_TF551/ai_TF551
//     Standard Inputs/MAIN.HNLT_CN.InnerCapillaryTubeMats.TS552.temperature_IN <-> K552A1_AI-2/2/ai_TF552/ai_TF552
//     Standard Inputs/MAIN.HNLT_CN.InnerCapillaryTubeMats.TS553.temperature_IN <-> K552A1_AI-2/2/ai_TF553/ai_TF553
//     Standard Inputs/MAIN.HNLT_CN.InnerCapillaryTubeMats.TS561.temperature_IN <-> K552A1_AI-2/2/ai_TF561/ai_TF561
//     Standard Inputs/MAIN.HNLT_CN.InnerCapillaryTubeMats.TS562.temperature_IN <-> K552A1_AI-2/2/ai_TF562/ai_TF562
//     Standard Inputs/MAIN.HNLT_CN.InnerCapillaryTubeMats.TS563.temperature_IN <-> K553A1_AI-1/2/ai_TF563/ai_TF563
//     Standard Inputs/MAIN.HNLT_CN.InnerCapillaryTubeMats.TS571.temperature_IN <-> K553A1_AI-1/2/ai_TF571/ai_TF571
//     Standard Inputs/MAIN.HNLT_CN.InnerCapillaryTubeMats.TS572.temperature_IN <-> K553A1_AI-1/2/ai_TF572/ai_TF572
//     Standard Inputs/MAIN.HNLT_CN.InnerCapillaryTubeMats.TS573.temperature_IN <-> K553A1_AI-1/2/ai_TF573/ai_TF573
//     Standard Inputs/MAIN.HNLT_CN.UnderfloorHeatingSystem.SV423.bStatusOff_IN <-> K533A1_BI/bi_SV423_Closed/bi_SV423_Closed
//     Standard Inputs/MAIN.HNLT_CN.UnderfloorHeatingSystem.SV424.bStatusOff_IN <-> K533A1_BI/bi_SV424_Closed/bi_SV424_Closed
//     Standard Inputs/MAIN.HNLT_CN.UnderfloorHeatingSystem.SV423.bStatusOn_IN <-> K533A1_BI/bi_SV423_Open/bi_SV423_Open
//     Standard Inputs/MAIN.HNLT_CN.UnderfloorHeatingSystem.SV424.bStatusOn_IN <-> K533A1_BI/bi_SV424_Open/bi_SV424_Open
//     Standard Outputs/.Dali_K522A1_DALI_OUT/nCtrl <-> K522A1_DALI/Channel 1/Kontrolle
//     Standard Outputs/.Dali_K522A1_DALI_OUT/nData <-> K522A1_DALI/Channel 1/Daten Aus
//     Standard Outputs/MAIN.Ambient.WeatherStation.KL6301_OUT @bit {16..184 step 8} <-> K523A1_EIB/Channel 1/Output Data {1..22}  (22 links)
//     Standard Outputs/MAIN.Ambient.WeatherStation.KL6301_OUT <-> K523A1_EIB/Channel 1/Parameter Control
//     Standard Outputs/MAIN.CN.CentralMachineCoolingSystem.SV100.bSetStatusOn_OUT <-> K540A1_BO/bo_SV100/bo_SV100
//     Standard Outputs/MAIN.CN.FlywheelMassStorageSystem.SV191.bSetStatusOn_OUT <-> K540A1_BO/bo_SV191/bo_SV191
//     Standard Outputs/MAIN.HNHT.CHP1System.CHP.bSetStatusOn_OUT <-> K542A1_BO/bo_CHP1/bo_CHP1_bSetStatusOn
//     Standard Outputs/MAIN.HNHT.CHP1System.CHP.nSetPoint_OUT <-> K570A1_AO-2/2/ao_CHP1_fSetPoint/ao_CHP1_fSetPoint
//     Standard Outputs/MAIN.HNHT.CHP2System.CHP.nSetPoint_OUT <-> K570A1_AO-2/2/ao_CHP2_fSetPoint/ao_CHP2_fSetPoint
//     Standard Outputs/MAIN.HNHT.CHP1System.SV32x.bSetStatusOn_OUT <-> K540A1_BO/bo_SV321/bo_SV321
//     Standard Outputs/MAIN.HNHT.CHP2System.SV32x.bSetStatusOn_OUT <-> K542A1_BO/bo_SV322/bo_SV322
//     Standard Outputs/MAIN.HNHT.CHP2System.CHP.bSetStatusOn_OUT <-> K542A1_BO/bo_CHP2/bo_CHP2
//     Standard Outputs/MAIN.HNHT.CentralMachineHeatingSystem.SV300.bSetStatusOn_OUT <-> K540A1_BO/bo_SV300/bo_SV300
//     Standard Outputs/MAIN.HNHT.CondensingBoilerSystem.SV331.bSetStatusOn_OUT <-> K542A1_BO/bo_SV331/bo_SV331
//     Standard Outputs/MAIN.HNHT.SV_SupplyAir.bSetStatusOn_OUT <-> K542A1_BO/bo_SV_SupplyAir_CHP/bo_SV_SupplyAir_CHP
//     Standard Outputs/MAIN.HNHT.StaticHeatingSystem.RV350.nSetPoint_OUT <-> K570A1_AO-1/2/ao_RV350/ao_RV350
//     Standard Outputs/MAIN.HNHT_CN.VentilationSystem.SV453.bSetStatusOn_OUT <-> K544A1_BO/bo_SV453/bo_SV453
//     Standard Outputs/MAIN.HNHT_CN.VentilationSystem.SV454.bSetStatusOn_OUT <-> K544A1_BO/bo_SV454/bo_SV454
//     Standard Outputs/MAIN.HNHT_HNLT.HeatExchanger1System.SV215.bSetStatusOn_OUT <-> K540A1_BO/bo_SV215/bo_SV215
//     Standard Outputs/MAIN.HNLT.DCSystem.SV245.bSetStatusOn_OUT <-> K540A1_BO/bo_SV245/bo_SV245
//     Standard Outputs/MAIN.HNLT.OuterCapillaryTubeMats.PU690.bSetStatusOn_OUT <-> K542A1_BO/bo_PU690/bo_PU690
//     Standard Outputs/MAIN.HNLT.OuterCapillaryTubeMats.RV600.nSetPoint_OUT <-> K572A1_AO-2/2/ao_RV600/ao_RV600
//     Standard Outputs/MAIN.HNLT.OuterCapillaryTubeMats.RV640.nSetPoint_OUT <-> K572A1_AO-2/2/ao_RV640/ao_RV640
//     Standard Outputs/MAIN.HNLT.OuterCapillaryTubeMats.RV660.nSetPoint_OUT <-> K573A1_AO-1/2/ao_RV660/ao_RV660
//     Standard Outputs/MAIN.HNLT.OuterCapillaryTubeMats.SV235.bSetStatusOn_OUT <-> K540A1_BO/bo_SV235/bo_SV235
//     Standard Outputs/MAIN.HNLT.OuterCapillaryTubeMats.SV605.bSetStatusOn_OUT <-> K542A1_BO/bo_SV605/bo_SV605
//     Standard Outputs/MAIN.HNLT_CN.HeatPumpSystem.HeatPump.bSetStatusOn_OUT <-> K544A1_BO/bo_HeatPump/bo_HeatPump
//     Standard Outputs/MAIN.HNLT_CN.HeatPumpSystem.SV146.bSetStatusOn_OUT <-> K544A1_BO/bo_SV146/bo_SV146
//     Standard Outputs/MAIN.HNLT_CN.HeatPumpSystem.SV246.bSetStatusOn_OUT <-> K544A1_BO/bo_SV246/bo_SV246
//     Standard Outputs/MAIN.HNLT_CN.InnerCapillaryTubeMats.RV500.nSetPoint_OUT <-> K571A1_AO-1/2/ao_RV500/ao_RV500
//     Standard Outputs/MAIN.HNLT_CN.InnerCapillaryTubeMats.RV541.nSetPoint_OUT <-> K571A1_AO-1/2/ao_RV541/ao_RV541
//     Standard Outputs/MAIN.HNLT_CN.InnerCapillaryTubeMats.RV542.nSetPoint_OUT <-> K571A1_AO-1/2/ao_RV542/ao_RV542
//     Standard Outputs/MAIN.HNLT_CN.InnerCapillaryTubeMats.RV543.nSetPoint_OUT <-> K571A1_AO-2/2/ao_RV543/ao_RV543
//     Standard Outputs/MAIN.HNLT_CN.InnerCapillaryTubeMats.RV551.nSetPoint_OUT <-> K571A1_AO-2/2/ao_RV551/ao_RV551
//     Standard Outputs/MAIN.HNLT_CN.InnerCapillaryTubeMats.RV552.nSetPoint_OUT <-> K571A1_AO-2/2/ao_RV552/ao_RV552
//     Standard Outputs/MAIN.HNLT_CN.InnerCapillaryTubeMats.RV553.nSetPoint_OUT <-> K571A1_AO-2/2/ao_RV553/ao_RV553
//     Standard Outputs/MAIN.HNLT_CN.InnerCapillaryTubeMats.RV561.nSetPoint_OUT <-> K572A1_AO-1/2/ao_RV561/ao_RV561
//     Standard Outputs/MAIN.HNLT_CN.InnerCapillaryTubeMats.RV562.nSetPoint_OUT <-> K572A1_AO-1/2/ao_RV562/ao_RV562
//     Standard Outputs/MAIN.HNLT_CN.InnerCapillaryTubeMats.RV563.nSetPoint_OUT <-> K572A1_AO-1/2/ao_RV563/ao_RV563
//     Standard Outputs/MAIN.HNLT_CN.InnerCapillaryTubeMats.RV571.nSetPoint_OUT <-> K572A1_AO-1/2/ao_RV571/ao_RV571
//     Standard Outputs/MAIN.HNLT_CN.InnerCapillaryTubeMats.RV572.nSetPoint_OUT <-> K572A1_AO-2/2/ao_RV572/ao_RV572
//     Standard Outputs/MAIN.HNLT_CN.InnerCapillaryTubeMats.RV573.nSetPoint_OUT <-> K572A1_AO-2/2/ao_RV573/ao_RV573
//     Standard Outputs/MAIN.HNLT_CN.InnerCapillaryTubeMats.SV505.bSetStatusOn_OUT <-> K542A1_BO/bo_SV505/bo_SV505
//     Standard Outputs/MAIN.HNLT_CN.InnerCapillaryTubeMats.SV_CN.bSetStatusOn_OUT <-> K542A1_BO/bo_SV_CN_HeatExchanger3/bo_SV_CN_HeatExchanger3
//     Standard Outputs/MAIN.HNLT_CN.InnerCapillaryTubeMats.SV_HNLT.bSetStatusOn_OUT <-> K542A1_BO/bo_SV_HNLT_HeatExchanger3/bo_SV_HNLT_HeatExchanger3
//     Standard Outputs/MAIN.HNLT_CN.UnderfloorHeatingSystem.RV425.nSetPoint_OUT <-> K570A1_AO-2/2/ao_RV425/ao_RV425
//     Standard Outputs/MAIN.HNLT_CN.UnderfloorHeatingSystem.SV423.bSetStatusOn_OUT <-> K542A1_BO/bo_SV423/bo_SV423
//     Standard Outputs/MAIN.HNLT_CN.UnderfloorHeatingSystem.SV424.bSetStatusOn_OUT <-> K542A1_BO/bo_SV424/bo_SV424
//   CP_5C7432/CP_5C7432 Instance <-> Device 10 (EtherCAT)/Term 64 (EK1100)/Box 55 (BK1250)
//     MBus_WZaehler_Task Inputs/.IN_WZaehler_Basement/D <-> Term 255 (KL6781)/Channel 1/Data In 0
//     MBus_WZaehler_Task Inputs/.IN_WZaehler_Basement/D @bit {8..168 step 8} <-> Term 255 (KL6781)/Channel 1/Data In {1..21}  (21 links)
//     MBus_WZaehler_Task Inputs/.IN_WZaehler_Basement/Status <-> Term 255 (KL6781)/Channel 1/Status
//     MBus_WZaehler_Task Outputs/.OUT_WZaehler_Basement/Ctrl <-> Term 255 (KL6781)/Channel 1/Ctrl
//     MBus_WZaehler_Task Outputs/.OUT_WZaehler_Basement/D <-> Term 255 (KL6781)/Channel 1/Data Out 0
//     MBus_WZaehler_Task Outputs/.OUT_WZaehler_Basement/D @bit {8..168 step 8} <-> Term 255 (KL6781)/Channel 1/Data Out {1..21}  (21 links)
//   CP_5C7432/CP_5C7432 Instance <-> Device 10 (EtherCAT)/Term 64 (EK1100)/Term 65 (EL3202-0010)
//     Standard Inputs/MAIN.HNHT.BufferStorage.MidTemperatureSensor.temperature_IN <-> ai_TF395_HNHT_MidTemperature/ai_TF395_MidTemperature
//     Standard Inputs/MAIN.HNHT.BufferStorage.UpperTemperatureSensor.temperature_IN <-> ai_TF395_HNHT_UpperTemperature/ai_TF395_HNHT_UpperTemperature
//   CP_5C7432/CP_5C7432 Instance <-> Device 10 (EtherCAT)/Term 64 (EK1100)/Term 66 (EL3202-0010)
//     Standard Inputs/MAIN.HNHT.BufferStorage.LowerTemperatureSensor.temperature_IN <-> ai_TF395_HNHT_LowerTemperature/ai_TF395_HNHT_LowerTemperature
//     Standard Inputs/MAIN.HNHT_HNLT.HeatPumpSystem.TS242.temperature_IN <-> ai_TF242_InletTemperature_HeatPump/ai_TF242_InletTemperature_HeatPump
//   CP_5C7432/CP_5C7432 Instance <-> Device 10 (EtherCAT)/Term 64 (EK1100)/Term 67 (EL3068)
//     Standard Inputs/MAIN.HNHT.VSIStorageSystem.SV305.nOperatingPoint_IN <-> ai_SV305/Value
//     Standard Inputs/MAIN.HNHT.VSIStorageSystem.SV306.nOperatingPoint_IN <-> ai_SV306/Value
//     Standard Inputs/MAIN.HNHT.VSIStorageSystem.SV307.nOperatingPoint_IN <-> ai_SV307/Value
//     Standard Inputs/MAIN.HNHT_HNLT.HeatPumpSystem.RV242.nOperatingPoint_IN <-> ai_RV242/ai_RV242
//     Standard Inputs/MAIN.HNHT_HNLT.HeatPumpSystem.RV342.nOperatingPoint_IN <-> ai_RV342/Value
//   CP_5C7432/CP_5C7432 Instance <-> Device 10 (EtherCAT)/Term 64 (EK1100)/Term 68 (EL4008)
//     Standard Outputs/MAIN.HNHT.CondensingBoilerSystem.CondensingBoiler.nSetPoint_OUT <-> ao_CondensingBoiler/ao_CondensingBoiler
//     Standard Outputs/MAIN.HNHT.VSIStorageSystem.SV305.nSetPoint_OUT <-> ao_SV305/Analog output
//     Standard Outputs/MAIN.HNHT.VSIStorageSystem.SV306.nSetPoint_OUT <-> ao_SV306/Analog output
//     Standard Outputs/MAIN.HNHT.VSIStorageSystem.SV307.nSetPoint_OUT <-> ao_SV307/Analog output
//     Standard Outputs/MAIN.HNHT_HNLT.HeatPumpSystem.HeatPump.nSetPoint_OUT <-> ao_HNHT_HeatPump/ao_HNHT_HeatPump
//     Standard Outputs/MAIN.HNHT_HNLT.HeatPumpSystem.RV242.nSetPoint_OUT <-> ao_RV242/ao_RV242
//     Standard Outputs/MAIN.HNHT_HNLT.HeatPumpSystem.RV342.nSetPoint_OUT <-> ao_RV342/ao_RV342
//   CP_5C7432/CP_5C7432 Instance <-> Device 10 (EtherCAT)/Term 64 (EK1100)/Term 69 (EL1809)
//     Standard Inputs/MAIN.HNHT.CondensingBoilerSystem.CondensingBoiler.bError_IN <-> bi_Error_CondensingBoiler/bi_Error_CondensingBoiler
//     Standard Inputs/MAIN.HNHT_HNLT.HeatPumpSystem.HeatPump.bError_IN <-> bi_Error_HeatPump_HNHT/bi_Error_HeatPump_HNHT
//   CP_5C7432/CP_5C7432 Instance <-> Device 10 (EtherCAT)/Term 64 (EK1100)/Term 70 (EL2809)
//     Standard Outputs/MAIN.HNHT.CondensingBoilerSystem.CondensingBoiler.bSetStatusOn_OUT <-> bo_CondensingBoiler/bo_CondensingBoiler
//     Standard Outputs/MAIN.HNHT_HNLT.HeatPumpSystem.HeatPump.bSetStatusOn_OUT <-> bo_HeatPump_HNHT/bo_HeatPump_HNHT
//     Standard Outputs/MAIN.HNHT_HNLT.HeatPumpSystem.SV_HNLT.bSetStatusOn_OUT <-> bo_HeatPump_HNHT_SV_HNLT_Open/bo_HeatPump_HNHT_SV_HNLT_Open
//   CP_5C7432/CP_5C7432 Instance <-> Device 2 (EL6731)/Box 1 (CIM/CIU 150 pump)
//     Standard Inputs/MAIN.HNLT.OuterCapillaryTubeMats.PU235.StatusModule_IN <-> StatusModule/Inputs/StatusModule_0_0
//     Standard Inputs/MAIN.HNLT.OuterCapillaryTubeMats.PU235.fActualSetpoint_IN <-> ActualSetpoint/Inputs/ActualSetpoint_0_0
//     Standard Inputs/MAIN.HNLT.OuterCapillaryTubeMats.PU235.fPowerElectric_IN <-> Power/Inputs/Power_0_0
//     Standard Inputs/MAIN.HNLT.OuterCapillaryTubeMats.PU235.fPowerThermal_IN <-> HeatPower/Inputs/HeatPower_0_0
//     Standard Inputs/MAIN.HNLT.OuterCapillaryTubeMats.PU235.fPressureDifference_IN <-> DiffPressure/Inputs/DiffPressure_0_0
//     Standard Inputs/MAIN.HNLT.OuterCapillaryTubeMats.PU235.fRotationalSpeed_IN <-> Speed/Inputs/Speed_0_0
//     Standard Inputs/MAIN.HNLT.OuterCapillaryTubeMats.PU235.fTemperatureDifference_IN <-> HeatDiffTemp/Inputs/HeatDiffTemp_0_0
//     Standard Inputs/MAIN.HNLT.OuterCapillaryTubeMats.PU235.fTemperatureExternal_IN <-> RemoteTemp2/Inputs/RemoteTemp2_0_0
//     Standard Inputs/MAIN.HNLT.OuterCapillaryTubeMats.PU235.fVolumeFlowRate_IN <-> VolumeFlow/Inputs/VolumeFlow_0_0
//     Standard Inputs/MAIN.HNLT.OuterCapillaryTubeMats.PU235.nAlarmCode_IN <-> FaultCode/Inputs/FaultCode_0_0
//     Standard Inputs/MAIN.HNLT.OuterCapillaryTubeMats.PU235.nWarningCode_IN <-> WarningCode/Inputs/WarningCode_0_0
//     Standard Inputs/MAIN.HNLT.OuterCapillaryTubeMats.PU235.stTemperatureInternal_Genibus_Reply <-> DirectDataReply/Inputs/DirectDataReply_0_0
//     Standard Outputs/MAIN.HNLT.OuterCapillaryTubeMats.PU235.ControlModule_OUT <-> ControlModule/Outputs/ControlModule_1_0
//     Standard Outputs/MAIN.HNLT.OuterCapillaryTubeMats.PU235.stTemperatureInternal_Genibus_Request <-> DirectDataRequest/Outputs/DirectDataRequest_1_0
//   CP_5C7432/CP_5C7432 Instance <-> Device 2 (EL6731)/Box 10 (CIM/CIU 150 pump)
//     Standard Inputs/MAIN.HNLT_CN.InnerCapillaryTubeMats.PU500.StatusModule_IN <-> StatusModule/Inputs/StatusModule_0_0
//     Standard Inputs/MAIN.HNLT_CN.InnerCapillaryTubeMats.PU500.fActualSetpoint_IN <-> ActualSetpoint/Inputs/ActualSetpoint_0_0
//     Standard Inputs/MAIN.HNLT_CN.InnerCapillaryTubeMats.PU500.fPowerElectric_IN <-> Power/Inputs/Power_0_0
//     Standard Inputs/MAIN.HNLT_CN.InnerCapillaryTubeMats.PU500.fPowerThermal_IN <-> HeatPower/Inputs/HeatPower_0_0
//     Standard Inputs/MAIN.HNLT_CN.InnerCapillaryTubeMats.PU500.fPressureDifference_IN <-> DiffPressure/Inputs/DiffPressure_0_0
//     Standard Inputs/MAIN.HNLT_CN.InnerCapillaryTubeMats.PU500.fRotationalSpeed_IN <-> Speed/Inputs/Speed_0_0
//     Standard Inputs/MAIN.HNLT_CN.InnerCapillaryTubeMats.PU500.fTemperatureDifference_IN <-> HeatDiffTemp/Inputs/HeatDiffTemp_0_0
//     Standard Inputs/MAIN.HNLT_CN.InnerCapillaryTubeMats.PU500.fTemperatureExternal_IN <-> RemoteTemp2/Inputs/RemoteTemp2_0_0
//     Standard Inputs/MAIN.HNLT_CN.InnerCapillaryTubeMats.PU500.fVolumeFlowRate_IN <-> VolumeFlow/Inputs/VolumeFlow_0_0
//     Standard Inputs/MAIN.HNLT_CN.InnerCapillaryTubeMats.PU500.nAlarmCode_IN <-> FaultCode/Inputs/FaultCode_0_0
//     Standard Inputs/MAIN.HNLT_CN.InnerCapillaryTubeMats.PU500.nWarningCode_IN <-> WarningCode/Inputs/WarningCode_0_0
//     Standard Inputs/MAIN.HNLT_CN.InnerCapillaryTubeMats.PU500.stTemperatureInternal_Genibus_Reply <-> DirectDataReply/Inputs/DirectDataReply_0_0
//     Standard Outputs/MAIN.HNLT_CN.InnerCapillaryTubeMats.PU500.ControlModule_OUT <-> ControlModule/Outputs/ControlModule_1_0
//     Standard Outputs/MAIN.HNLT_CN.InnerCapillaryTubeMats.PU500.stTemperatureInternal_Genibus_Request <-> DirectDataRequest/Outputs/DirectDataRequest_1_0
//   CP_5C7432/CP_5C7432 Instance <-> Device 2 (EL6731)/Box 11 (CIM/CIU 150 pump)
//     Standard Inputs/MAIN.HNLT_CN.UnderfloorHeatingSystem.PU425.StatusModule_IN <-> StatusModule/Inputs/StatusModule_0_0
//     Standard Inputs/MAIN.HNLT_CN.UnderfloorHeatingSystem.PU425.fActualSetpoint_IN <-> ActualSetpoint/Inputs/ActualSetpoint_0_0
//     Standard Inputs/MAIN.HNLT_CN.UnderfloorHeatingSystem.PU425.fPowerElectric_IN <-> Power/Inputs/Power_0_0
//     Standard Inputs/MAIN.HNLT_CN.UnderfloorHeatingSystem.PU425.fPowerThermal_IN <-> HeatPower/Inputs/HeatPower_0_0
//     Standard Inputs/MAIN.HNLT_CN.UnderfloorHeatingSystem.PU425.fPressureDifference_IN <-> DiffPressure/Inputs/DiffPressure_0_0
//     Standard Inputs/MAIN.HNLT_CN.UnderfloorHeatingSystem.PU425.fRotationalSpeed_IN <-> Speed/Inputs/Speed_0_0
//     Standard Inputs/MAIN.HNLT_CN.UnderfloorHeatingSystem.PU425.fTemperatureDifference_IN <-> HeatDiffTemp/Inputs/HeatDiffTemp_0_0
//     Standard Inputs/MAIN.HNLT_CN.UnderfloorHeatingSystem.PU425.fTemperatureExternal_IN <-> RemoteTemp2/Inputs/RemoteTemp2_0_0
//     Standard Inputs/MAIN.HNLT_CN.UnderfloorHeatingSystem.PU425.fVolumeFlowRate_IN <-> VolumeFlow/Inputs/VolumeFlow_0_0
//     Standard Inputs/MAIN.HNLT_CN.UnderfloorHeatingSystem.PU425.nAlarmCode_IN <-> FaultCode/Inputs/FaultCode_0_0
//     Standard Inputs/MAIN.HNLT_CN.UnderfloorHeatingSystem.PU425.nWarningCode_IN <-> WarningCode/Inputs/WarningCode_0_0
//     Standard Inputs/MAIN.HNLT_CN.UnderfloorHeatingSystem.PU425.stTemperatureInternal_Genibus_Reply <-> DirectDataReply/Inputs/DirectDataReply_0_0
//     Standard Outputs/MAIN.HNLT_CN.UnderfloorHeatingSystem.PU425.ControlModule_OUT <-> ControlModule/Outputs/ControlModule_1_0
//     Standard Outputs/MAIN.HNLT_CN.UnderfloorHeatingSystem.PU425.stTemperatureInternal_Genibus_Request <-> DirectDataRequest/Outputs/DirectDataRequest_1_0
//   CP_5C7432/CP_5C7432 Instance <-> Device 2 (EL6731)/Box 13 (CIM/CIU 150 pump)
//     Standard Inputs/MAIN.HNLT_CN.InnerCapillaryTubeMats.PU405.StatusModule_IN <-> StatusModule/Inputs/StatusModule_0_0
//     Standard Inputs/MAIN.HNLT_CN.InnerCapillaryTubeMats.PU405.fActualSetpoint_IN <-> ActualSetpoint/Inputs/ActualSetpoint_0_0
//     Standard Inputs/MAIN.HNLT_CN.InnerCapillaryTubeMats.PU405.fPowerElectric_IN <-> Power/Inputs/Power_0_0
//     Standard Inputs/MAIN.HNLT_CN.InnerCapillaryTubeMats.PU405.fPowerThermal_IN <-> HeatPower/Inputs/HeatPower_0_0
//     Standard Inputs/MAIN.HNLT_CN.InnerCapillaryTubeMats.PU405.fPressureDifference_IN <-> DiffPressure/Inputs/DiffPressure_0_0
//     Standard Inputs/MAIN.HNLT_CN.InnerCapillaryTubeMats.PU405.fRotationalSpeed_IN <-> Speed/Inputs/Speed_0_0
//     Standard Inputs/MAIN.HNLT_CN.InnerCapillaryTubeMats.PU405.fTemperatureDifference_IN <-> HeatDiffTemp/Inputs/HeatDiffTemp_0_0
//     Standard Inputs/MAIN.HNLT_CN.InnerCapillaryTubeMats.PU405.fTemperatureExternal_IN <-> RemoteTemp2/Inputs/RemoteTemp2_0_0
//     Standard Inputs/MAIN.HNLT_CN.InnerCapillaryTubeMats.PU405.fVolumeFlowRate_IN <-> VolumeFlow/Inputs/VolumeFlow_0_0
//     Standard Inputs/MAIN.HNLT_CN.InnerCapillaryTubeMats.PU405.nAlarmCode_IN <-> FaultCode/Inputs/FaultCode_0_0
//     Standard Inputs/MAIN.HNLT_CN.InnerCapillaryTubeMats.PU405.nWarningCode_IN <-> WarningCode/Inputs/WarningCode_0_0
//     Standard Inputs/MAIN.HNLT_CN.InnerCapillaryTubeMats.PU405.stTemperatureInternal_Genibus_Reply <-> DirectDataReply/Inputs/DirectDataReply_0_0
//     Standard Outputs/MAIN.HNLT_CN.InnerCapillaryTubeMats.PU405.ControlModule_OUT <-> ControlModule/Outputs/ControlModule_1_0
//     Standard Outputs/MAIN.HNLT_CN.InnerCapillaryTubeMats.PU405.stTemperatureInternal_Genibus_Request <-> DirectDataRequest/Outputs/DirectDataRequest_1_0
//   CP_5C7432/CP_5C7432 Instance <-> Device 2 (EL6731)/Box 14 (CIM/CIU 150 pump)
//     Standard Inputs/MAIN.HNLT.CompressorSystem.PU251.StatusModule_IN <-> StatusModule/Inputs/StatusModule_0_0
//     Standard Inputs/MAIN.HNLT.CompressorSystem.PU251.fActualSetpoint_IN <-> ActualSetpoint/Inputs/ActualSetpoint_0_0
//     Standard Inputs/MAIN.HNLT.CompressorSystem.PU251.fPowerElectric_IN <-> Power/Inputs/Power_0_0
//     Standard Inputs/MAIN.HNLT.CompressorSystem.PU251.fPowerThermal_IN <-> HeatPower/Inputs/HeatPower_0_0
//     Standard Inputs/MAIN.HNLT.CompressorSystem.PU251.fPressureDifference_IN <-> DiffPressure/Inputs/DiffPressure_0_0
//     Standard Inputs/MAIN.HNLT.CompressorSystem.PU251.fRotationalSpeed_IN <-> Speed/Inputs/Speed_0_0
//     Standard Inputs/MAIN.HNLT.CompressorSystem.PU251.fTemperatureDifference_IN <-> HeatDiffTemp/Inputs/HeatDiffTemp_0_0
//     Standard Inputs/MAIN.HNLT.CompressorSystem.PU251.fTemperatureExternal_IN <-> RemoteTemp2/Inputs/RemoteTemp2_0_0
//     Standard Inputs/MAIN.HNLT.CompressorSystem.PU251.fVolumeFlowRate_IN <-> VolumeFlow/Inputs/VolumeFlow_0_0
//     Standard Inputs/MAIN.HNLT.CompressorSystem.PU251.nAlarmCode_IN <-> FaultCode/Inputs/FaultCode_0_0
//     Standard Inputs/MAIN.HNLT.CompressorSystem.PU251.nWarningCode_IN <-> WarningCode/Inputs/WarningCode_0_0
//     Standard Inputs/MAIN.HNLT.CompressorSystem.PU251.stTemperatureInternal_Genibus_Reply <-> DirectDataReply/Inputs/DirectDataReply_0_0
//     Standard Outputs/MAIN.HNLT.CompressorSystem.PU251.ControlModule_OUT <-> ControlModule/Outputs/ControlModule_1_0
//     Standard Outputs/MAIN.HNLT.CompressorSystem.PU251.stTemperatureInternal_Genibus_Request <-> DirectDataRequest/Outputs/DirectDataRequest_1_0
//   CP_5C7432/CP_5C7432 Instance <-> Device 2 (EL6731)/Box 15 (CIM/CIU 150 pump)
//     Standard Inputs/MAIN.HNHT_CN.VentilationSystem.PU455.StatusModule_IN <-> StatusModule/Inputs/StatusModule_0_0
//     Standard Inputs/MAIN.HNHT_CN.VentilationSystem.PU455.fActualSetpoint_IN <-> ActualSetpoint/Inputs/ActualSetpoint_0_0
//     Standard Inputs/MAIN.HNHT_CN.VentilationSystem.PU455.fPowerElectric_IN <-> Power/Inputs/Power_0_0
//     Standard Inputs/MAIN.HNHT_CN.VentilationSystem.PU455.fPowerThermal_IN <-> HeatPower/Inputs/HeatPower_0_0
//     Standard Inputs/MAIN.HNHT_CN.VentilationSystem.PU455.fPressureDifference_IN <-> DiffPressure/Inputs/DiffPressure_0_0
//     Standard Inputs/MAIN.HNHT_CN.VentilationSystem.PU455.fRotationalSpeed_IN <-> Speed/Inputs/Speed_0_0
//     Standard Inputs/MAIN.HNHT_CN.VentilationSystem.PU455.fTemperatureDifference_IN <-> HeatDiffTemp/Inputs/HeatDiffTemp_0_0
//     Standard Inputs/MAIN.HNHT_CN.VentilationSystem.PU455.fTemperatureExternal_IN <-> RemoteTemp2/Inputs/RemoteTemp2_0_0
//     Standard Inputs/MAIN.HNHT_CN.VentilationSystem.PU455.fVolumeFlowRate_IN <-> VolumeFlow/Inputs/VolumeFlow_0_0
//     Standard Inputs/MAIN.HNHT_CN.VentilationSystem.PU455.nAlarmCode_IN <-> FaultCode/Inputs/FaultCode_0_0
//     Standard Inputs/MAIN.HNHT_CN.VentilationSystem.PU455.nWarningCode_IN <-> WarningCode/Inputs/WarningCode_0_0
//     Standard Inputs/MAIN.HNHT_CN.VentilationSystem.PU455.stTemperatureInternal_Genibus_Reply <-> DirectDataReply/Inputs/DirectDataReply_0_0
//     Standard Outputs/MAIN.HNHT_CN.VentilationSystem.PU455.stTemperatureInternal_Genibus_Request <-> DirectDataRequest/Outputs/DirectDataRequest_1_0
//   CP_5C7432/CP_5C7432 Instance <-> Device 2 (EL6731)/Box 16 (CIM/CIU 150 pump)
//     Standard Inputs/MAIN.HNHT.StaticHeatingSystem.PU350.StatusModule_IN <-> StatusModule/Inputs/StatusModule_0_0
//     Standard Inputs/MAIN.HNHT.StaticHeatingSystem.PU350.fActualSetpoint_IN <-> ActualSetpoint/Inputs/ActualSetpoint_0_0
//     Standard Inputs/MAIN.HNHT.StaticHeatingSystem.PU350.fPowerElectric_IN <-> Power/Inputs/Power_0_0
//     Standard Inputs/MAIN.HNHT.StaticHeatingSystem.PU350.fPowerThermal_IN <-> HeatPower/Inputs/HeatPower_0_0
//     Standard Inputs/MAIN.HNHT.StaticHeatingSystem.PU350.fPressureDifference_IN <-> DiffPressure/Inputs/DiffPressure_0_0
//     Standard Inputs/MAIN.HNHT.StaticHeatingSystem.PU350.fRotationalSpeed_IN <-> Speed/Inputs/Speed_0_0
//     Standard Inputs/MAIN.HNHT.StaticHeatingSystem.PU350.fTemperatureDifference_IN <-> HeatDiffTemp/Inputs/HeatDiffTemp_0_0
//     Standard Inputs/MAIN.HNHT.StaticHeatingSystem.PU350.fTemperatureExternal_IN <-> RemoteTemp2/Inputs/RemoteTemp2_0_0
//     Standard Inputs/MAIN.HNHT.StaticHeatingSystem.PU350.fVolumeFlowRate_IN <-> VolumeFlow/Inputs/VolumeFlow_0_0
//     Standard Inputs/MAIN.HNHT.StaticHeatingSystem.PU350.nAlarmCode_IN <-> FaultCode/Inputs/FaultCode_0_0
//     Standard Inputs/MAIN.HNHT.StaticHeatingSystem.PU350.nWarningCode_IN <-> WarningCode/Inputs/WarningCode_0_0
//     Standard Inputs/MAIN.HNHT.StaticHeatingSystem.PU350.stTemperatureInternal_Genibus_Reply <-> DirectDataReply/Inputs/DirectDataReply_0_0
//     Standard Outputs/MAIN.HNHT.StaticHeatingSystem.PU350.ControlModule_OUT <-> ControlModule/Outputs/ControlModule_1_0
//     Standard Outputs/MAIN.HNHT.StaticHeatingSystem.PU350.stTemperatureInternal_Genibus_Request <-> DirectDataRequest/Outputs/DirectDataRequest_1_0
//   CP_5C7432/CP_5C7432 Instance <-> Device 2 (EL6731)/Box 17 (CIM/CIU 150 pump)
//     Standard Inputs/MAIN.CN.FlywheelMassStorageSystem.PU191.StatusModule_IN <-> StatusModule/Inputs/StatusModule_0_0
//     Standard Inputs/MAIN.CN.FlywheelMassStorageSystem.PU191.fActualSetpoint_IN <-> ActualSetpoint/Inputs/ActualSetpoint_0_0
//     Standard Inputs/MAIN.CN.FlywheelMassStorageSystem.PU191.fPowerElectric_IN <-> Power/Inputs/Power_0_0
//     Standard Inputs/MAIN.CN.FlywheelMassStorageSystem.PU191.fPowerThermal_IN <-> HeatPower/Inputs/HeatPower_0_0
//     Standard Inputs/MAIN.CN.FlywheelMassStorageSystem.PU191.fPressureDifference_IN <-> DiffPressure/Inputs/DiffPressure_0_0
//     Standard Inputs/MAIN.CN.FlywheelMassStorageSystem.PU191.fRotationalSpeed_IN <-> Speed/Inputs/Speed_0_0
//     Standard Inputs/MAIN.CN.FlywheelMassStorageSystem.PU191.fTemperatureDifference_IN <-> HeatDiffTemp/Inputs/HeatDiffTemp_0_0
//     Standard Inputs/MAIN.CN.FlywheelMassStorageSystem.PU191.fTemperatureExternal_IN <-> RemoteTemp2/Inputs/RemoteTemp2_0_0
//     Standard Inputs/MAIN.CN.FlywheelMassStorageSystem.PU191.fVolumeFlowRate_IN <-> VolumeFlow/Inputs/VolumeFlow_0_0
//     Standard Inputs/MAIN.CN.FlywheelMassStorageSystem.PU191.nAlarmCode_IN <-> FaultCode/Inputs/FaultCode_0_0
//     Standard Inputs/MAIN.CN.FlywheelMassStorageSystem.PU191.nWarningCode_IN <-> WarningCode/Inputs/WarningCode_0_0
//     Standard Inputs/MAIN.CN.FlywheelMassStorageSystem.PU191.stTemperatureInternal_Genibus_Reply <-> DirectDataReply/Inputs/DirectDataReply_0_0
//     Standard Outputs/MAIN.CN.FlywheelMassStorageSystem.PU191.ControlModule_OUT <-> ControlModule/Outputs/ControlModule_1_0
//     Standard Outputs/MAIN.CN.FlywheelMassStorageSystem.PU191.stTemperatureInternal_Genibus_Request <-> DirectDataRequest/Outputs/DirectDataRequest_1_0
//   CP_5C7432/CP_5C7432 Instance <-> Device 2 (EL6731)/Box 20 (CIM/CIU 150 pump)
//     Standard Inputs/MAIN.HNHT.VSIStorageSystem.PU305.StatusModule_IN <-> StatusModule/Inputs/StatusModule_0_0
//     Standard Inputs/MAIN.HNHT.VSIStorageSystem.PU305.fActualSetpoint_IN <-> ActualSetpoint/Inputs/ActualSetpoint_0_0
//     Standard Inputs/MAIN.HNHT.VSIStorageSystem.PU305.fPowerElectric_IN <-> Power/Inputs/Power_0_0
//     Standard Inputs/MAIN.HNHT.VSIStorageSystem.PU305.fPowerThermal_IN <-> HeatPower/Inputs/HeatPower_0_0
//     Standard Inputs/MAIN.HNHT.VSIStorageSystem.PU305.fPressureDifference_IN <-> DiffPressure/Inputs/DiffPressure_0_0
//     Standard Inputs/MAIN.HNHT.VSIStorageSystem.PU305.fRotationalSpeed_IN <-> Speed/Inputs/Speed_0_0
//     Standard Inputs/MAIN.HNHT.VSIStorageSystem.PU305.fTemperatureDifference_IN <-> HeatDiffTemp/Inputs/HeatDiffTemp_0_0
//     Standard Inputs/MAIN.HNHT.VSIStorageSystem.PU305.fTemperatureExternal_IN <-> RemoteTemp2/Inputs/RemoteTemp2_0_0
//     Standard Inputs/MAIN.HNHT.VSIStorageSystem.PU305.fVolumeFlowRate_IN <-> VolumeFlow/Inputs/VolumeFlow_0_0
//     Standard Inputs/MAIN.HNHT.VSIStorageSystem.PU305.nAlarmCode_IN <-> FaultCode/Inputs/FaultCode_0_0
//     Standard Inputs/MAIN.HNHT.VSIStorageSystem.PU305.nWarningCode_IN <-> WarningCode/Inputs/WarningCode_0_0
//     Standard Inputs/MAIN.HNHT.VSIStorageSystem.PU305.stTemperatureInternal_Genibus_Reply <-> DirectDataReply/Inputs/DirectDataReply_0_0
//     Standard Outputs/MAIN.HNHT.VSIStorageSystem.PU305.ControlModule_OUT <-> ControlModule/Outputs/ControlModule_1_0
//     Standard Outputs/MAIN.HNHT.VSIStorageSystem.PU305.stTemperatureInternal_Genibus_Request <-> DirectDataRequest/Outputs/DirectDataRequest_1_0
//   CP_5C7432/CP_5C7432 Instance <-> Device 2 (EL6731)/Box 21 (CIM/CIU 150 pump)
//     Standard Inputs/MAIN.HNHT.VSIStorageSystem.PU306.StatusModule_IN <-> StatusModule/Inputs/StatusModule_0_0
//     Standard Inputs/MAIN.HNHT.VSIStorageSystem.PU306.fActualSetpoint_IN <-> ActualSetpoint/Inputs/ActualSetpoint_0_0
//     Standard Inputs/MAIN.HNHT.VSIStorageSystem.PU306.fPowerElectric_IN <-> Power/Inputs/Power_0_0
//     Standard Inputs/MAIN.HNHT.VSIStorageSystem.PU306.fPowerThermal_IN <-> HeatPower/Inputs/HeatPower_0_0
//     Standard Inputs/MAIN.HNHT.VSIStorageSystem.PU306.fPressureDifference_IN <-> DiffPressure/Inputs/DiffPressure_0_0
//     Standard Inputs/MAIN.HNHT.VSIStorageSystem.PU306.fRotationalSpeed_IN <-> Speed/Inputs/Speed_0_0
//     Standard Inputs/MAIN.HNHT.VSIStorageSystem.PU306.fTemperatureDifference_IN <-> HeatDiffTemp/Inputs/HeatDiffTemp_0_0
//     Standard Inputs/MAIN.HNHT.VSIStorageSystem.PU306.fTemperatureExternal_IN <-> RemoteTemp2/Inputs/RemoteTemp2_0_0
//     Standard Inputs/MAIN.HNHT.VSIStorageSystem.PU306.fVolumeFlowRate_IN <-> VolumeFlow/Inputs/VolumeFlow_0_0
//     Standard Inputs/MAIN.HNHT.VSIStorageSystem.PU306.nAlarmCode_IN <-> FaultCode/Inputs/FaultCode_0_0
//     Standard Inputs/MAIN.HNHT.VSIStorageSystem.PU306.nWarningCode_IN <-> WarningCode/Inputs/WarningCode_0_0
//     Standard Inputs/MAIN.HNHT.VSIStorageSystem.PU306.stTemperatureInternal_Genibus_Reply <-> DirectDataReply/Inputs/DirectDataReply_0_0
//     Standard Outputs/MAIN.HNHT.VSIStorageSystem.PU306.ControlModule_OUT <-> ControlModule/Outputs/ControlModule_1_0
//     Standard Outputs/MAIN.HNHT.VSIStorageSystem.PU306.stTemperatureInternal_Genibus_Request <-> DirectDataRequest/Outputs/DirectDataRequest_1_0
//   CP_5C7432/CP_5C7432 Instance <-> Device 2 (EL6731)/Box 22 (CIM/CIU 150 pump)
//     Standard Inputs/MAIN.HNHT_HNLT.HeatPumpSystem.PU242.StatusModule_IN <-> StatusModule/Inputs/StatusModule_0_0
//     Standard Inputs/MAIN.HNHT_HNLT.HeatPumpSystem.PU242.fActualSetpoint_IN <-> ActualSetpoint/Inputs/ActualSetpoint_0_0
//     Standard Inputs/MAIN.HNHT_HNLT.HeatPumpSystem.PU242.fPowerElectric_IN <-> Power/Inputs/Power_0_0
//     Standard Inputs/MAIN.HNHT_HNLT.HeatPumpSystem.PU242.fPowerThermal_IN <-> HeatPower/Inputs/HeatPower_0_0
//     Standard Inputs/MAIN.HNHT_HNLT.HeatPumpSystem.PU242.fPressureDifference_IN <-> DiffPressure/Inputs/DiffPressure_0_0
//     Standard Inputs/MAIN.HNHT_HNLT.HeatPumpSystem.PU242.fRotationalSpeed_IN <-> Speed/Inputs/Speed_0_0
//     Standard Inputs/MAIN.HNHT_HNLT.HeatPumpSystem.PU242.fTemperatureDifference_IN <-> HeatDiffTemp/Inputs/HeatDiffTemp_0_0
//     Standard Inputs/MAIN.HNHT_HNLT.HeatPumpSystem.PU242.fTemperatureExternal_IN <-> RemoteTemp2/Inputs/RemoteTemp2_0_0
//     Standard Inputs/MAIN.HNHT_HNLT.HeatPumpSystem.PU242.fVolumeFlowRate_IN <-> VolumeFlow/Inputs/VolumeFlow_0_0
//     Standard Inputs/MAIN.HNHT_HNLT.HeatPumpSystem.PU242.nAlarmCode_IN <-> FaultCode/Inputs/FaultCode_0_0
//     Standard Inputs/MAIN.HNHT_HNLT.HeatPumpSystem.PU242.nWarningCode_IN <-> WarningCode/Inputs/WarningCode_0_0
//     Standard Inputs/MAIN.HNHT_HNLT.HeatPumpSystem.PU242.stTemperatureInternal_Genibus_Reply <-> DirectDataReply/Inputs/DirectDataReply_0_0
//     Standard Outputs/MAIN.HNHT_HNLT.HeatPumpSystem.PU242.ControlModule_OUT <-> ControlModule/Outputs/ControlModule_1_0
//     Standard Outputs/MAIN.HNHT_HNLT.HeatPumpSystem.PU242.stTemperatureInternal_Genibus_Request <-> DirectDataRequest/Outputs/DirectDataRequest_1_0
//   CP_5C7432/CP_5C7432 Instance <-> Device 2 (EL6731)/Box 3 (CIM/CIU 150 pump)
//     Standard Inputs/MAIN.HNHT_HNLT.HeatExchanger1System.PU215.StatusModule_IN <-> StatusModule/Inputs/StatusModule_0_0
//     Standard Inputs/MAIN.HNHT_HNLT.HeatExchanger1System.PU215.fActualSetpoint_IN <-> ActualSetpoint/Inputs/ActualSetpoint_0_0
//     Standard Inputs/MAIN.HNHT_HNLT.HeatExchanger1System.PU215.fPowerElectric_IN <-> Power/Inputs/Power_0_0
//     Standard Inputs/MAIN.HNHT_HNLT.HeatExchanger1System.PU215.fPowerThermal_IN <-> HeatPower/Inputs/HeatPower_0_0
//     Standard Inputs/MAIN.HNHT_HNLT.HeatExchanger1System.PU215.fPressureDifference_IN <-> DiffPressure/Inputs/DiffPressure_0_0
//     Standard Inputs/MAIN.HNHT_HNLT.HeatExchanger1System.PU215.fRotationalSpeed_IN <-> Speed/Inputs/Speed_0_0
//     Standard Inputs/MAIN.HNHT_HNLT.HeatExchanger1System.PU215.fTemperatureDifference_IN <-> HeatDiffTemp/Inputs/HeatDiffTemp_0_0
//     Standard Inputs/MAIN.HNHT_HNLT.HeatExchanger1System.PU215.fTemperatureExternal_IN <-> RemoteTemp2/Inputs/RemoteTemp2_0_0
//     Standard Inputs/MAIN.HNHT_HNLT.HeatExchanger1System.PU215.fVolumeFlowRate_IN <-> VolumeFlow/Inputs/VolumeFlow_0_0
//     Standard Inputs/MAIN.HNHT_HNLT.HeatExchanger1System.PU215.nAlarmCode_IN <-> FaultCode/Inputs/FaultCode_0_0
//     Standard Inputs/MAIN.HNHT_HNLT.HeatExchanger1System.PU215.nWarningCode_IN <-> WarningCode/Inputs/WarningCode_0_0
//     Standard Inputs/MAIN.HNHT_HNLT.HeatExchanger1System.PU215.stTemperatureInternal_Genibus_Reply <-> DirectDataReply/Inputs/DirectDataReply_0_0
//     Standard Outputs/MAIN.HNHT_HNLT.HeatExchanger1System.PU215.ControlModule_OUT <-> ControlModule/Outputs/ControlModule_1_0
//     Standard Outputs/MAIN.HNHT_HNLT.HeatExchanger1System.PU215.stTemperatureInternal_Genibus_Request <-> DirectDataRequest/Outputs/DirectDataRequest_1_0
//   CP_5C7432/CP_5C7432 Instance <-> Device 2 (EL6731)/Box 4 (CIM/CIU 150 pump)
//     Standard Inputs/MAIN.HNHT_HNLT.HeatExchanger1System.PU315.StatusModule_IN <-> StatusModule/Inputs/StatusModule_0_0
//     Standard Inputs/MAIN.HNHT_HNLT.HeatExchanger1System.PU315.fActualSetpoint_IN <-> ActualSetpoint/Inputs/ActualSetpoint_0_0
//     Standard Inputs/MAIN.HNHT_HNLT.HeatExchanger1System.PU315.fPowerElectric_IN <-> Power/Inputs/Power_0_0
//     Standard Inputs/MAIN.HNHT_HNLT.HeatExchanger1System.PU315.fPowerThermal_IN <-> HeatPower/Inputs/HeatPower_0_0
//     Standard Inputs/MAIN.HNHT_HNLT.HeatExchanger1System.PU315.fPressureDifference_IN <-> DiffPressure/Inputs/DiffPressure_0_0
//     Standard Inputs/MAIN.HNHT_HNLT.HeatExchanger1System.PU315.fRotationalSpeed_IN <-> Speed/Inputs/Speed_0_0
//     Standard Inputs/MAIN.HNHT_HNLT.HeatExchanger1System.PU315.fTemperatureDifference_IN <-> HeatDiffTemp/Inputs/HeatDiffTemp_0_0
//     Standard Inputs/MAIN.HNHT_HNLT.HeatExchanger1System.PU315.fTemperatureExternal_IN <-> RemoteTemp2/Inputs/RemoteTemp2_0_0
//     Standard Inputs/MAIN.HNHT_HNLT.HeatExchanger1System.PU315.fVolumeFlowRate_IN <-> VolumeFlow/Inputs/VolumeFlow_0_0
//     Standard Inputs/MAIN.HNHT_HNLT.HeatExchanger1System.PU315.nAlarmCode_IN <-> FaultCode/Inputs/FaultCode_0_0
//     Standard Inputs/MAIN.HNHT_HNLT.HeatExchanger1System.PU315.nWarningCode_IN <-> WarningCode/Inputs/WarningCode_0_0
//     Standard Inputs/MAIN.HNHT_HNLT.HeatExchanger1System.PU315.stTemperatureInternal_Genibus_Reply <-> DirectDataReply/Inputs/DirectDataReply_0_0
//     Standard Outputs/MAIN.HNHT_HNLT.HeatExchanger1System.PU315.ControlModule_OUT <-> ControlModule/Outputs/ControlModule_1_0
//     Standard Outputs/MAIN.HNHT_HNLT.HeatExchanger1System.PU315.stTemperatureInternal_Genibus_Request <-> DirectDataRequest/Outputs/DirectDataRequest_1_0
//   CP_5C7432/CP_5C7432 Instance <-> Device 2 (EL6731)/Box 5 (CIM/CIU 150 pump)
//     Standard Inputs/MAIN.HNHT.CHP2System.PU32x.StatusModule_IN <-> StatusModule/Inputs/StatusModule_0_0
//     Standard Inputs/MAIN.HNHT.CHP2System.PU32x.fActualSetpoint_IN <-> ActualSetpoint/Inputs/ActualSetpoint_0_0
//     Standard Inputs/MAIN.HNHT.CHP2System.PU32x.fPowerElectric_IN <-> Power/Inputs/Power_0_0
//     Standard Inputs/MAIN.HNHT.CHP2System.PU32x.fPowerThermal_IN <-> HeatPower/Inputs/HeatPower_0_0
//     Standard Inputs/MAIN.HNHT.CHP2System.PU32x.fPressureDifference_IN <-> DiffPressure/Inputs/DiffPressure_0_0
//     Standard Inputs/MAIN.HNHT.CHP2System.PU32x.fRotationalSpeed_IN <-> Speed/Inputs/Speed_0_0
//     Standard Inputs/MAIN.HNHT.CHP2System.PU32x.fTemperatureDifference_IN <-> HeatDiffTemp/Inputs/HeatDiffTemp_0_0
//     Standard Inputs/MAIN.HNHT.CHP2System.PU32x.fTemperatureExternal_IN <-> RemoteTemp2/Inputs/RemoteTemp2_0_0
//     Standard Inputs/MAIN.HNHT.CHP2System.PU32x.fVolumeFlowRate_IN <-> VolumeFlow/Inputs/VolumeFlow_0_0
//     Standard Inputs/MAIN.HNHT.CHP2System.PU32x.nAlarmCode_IN <-> FaultCode/Inputs/FaultCode_0_0
//     Standard Inputs/MAIN.HNHT.CHP2System.PU32x.nWarningCode_IN <-> WarningCode/Inputs/WarningCode_0_0
//     Standard Inputs/MAIN.HNHT.CHP2System.PU32x.stTemperatureInternal_Genibus_Reply <-> DirectDataReply/Inputs/DirectDataReply_0_0
//     Standard Outputs/MAIN.HNHT.CHP2System.PU32x.ControlModule_OUT <-> ControlModule/Outputs/ControlModule_1_0
//     Standard Outputs/MAIN.HNHT.CHP2System.PU32x.stTemperatureInternal_Genibus_Request <-> DirectDataRequest/Outputs/DirectDataRequest_1_0
//   CP_5C7432/CP_5C7432 Instance <-> Device 2 (EL6731)/Box 6 (CIM/CIU 150 pump)
//     Standard Inputs/MAIN.HNHT.CHP1System.PU32x.StatusModule_IN <-> StatusModule/Inputs/StatusModule_0_0
//     Standard Inputs/MAIN.HNHT.CHP1System.PU32x.fActualSetpoint_IN <-> ActualSetpoint/Inputs/ActualSetpoint_0_0
//     Standard Inputs/MAIN.HNHT.CHP1System.PU32x.fPowerElectric_IN <-> Power/Inputs/Power_0_0
//     Standard Inputs/MAIN.HNHT.CHP1System.PU32x.fPowerThermal_IN <-> HeatPower/Inputs/HeatPower_0_0
//     Standard Inputs/MAIN.HNHT.CHP1System.PU32x.fPressureDifference_IN <-> DiffPressure/Inputs/DiffPressure_0_0
//     Standard Inputs/MAIN.HNHT.CHP1System.PU32x.fRotationalSpeed_IN <-> Speed/Inputs/Speed_0_0
//     Standard Inputs/MAIN.HNHT.CHP1System.PU32x.fTemperatureDifference_IN <-> HeatDiffTemp/Inputs/HeatDiffTemp_0_0
//     Standard Inputs/MAIN.HNHT.CHP1System.PU32x.fTemperatureExternal_IN <-> RemoteTemp2/Inputs/RemoteTemp2_0_0
//     Standard Inputs/MAIN.HNHT.CHP1System.PU32x.fVolumeFlowRate_IN <-> VolumeFlow/Inputs/VolumeFlow_0_0
//     Standard Inputs/MAIN.HNHT.CHP1System.PU32x.nAlarmCode_IN <-> FaultCode/Inputs/FaultCode_0_0
//     Standard Inputs/MAIN.HNHT.CHP1System.PU32x.nWarningCode_IN <-> WarningCode/Inputs/WarningCode_0_0
//     Standard Inputs/MAIN.HNHT.CHP1System.PU32x.stTemperatureInternal_Genibus_Reply <-> DirectDataReply/Inputs/DirectDataReply_0_0
//     Standard Outputs/MAIN.HNHT.CHP1System.PU32x.ControlModule_OUT <-> ControlModule/Outputs/ControlModule_1_0
//     Standard Outputs/MAIN.HNHT.CHP1System.PU32x.stTemperatureInternal_Genibus_Request <-> DirectDataRequest/Outputs/DirectDataRequest_1_0
//   CP_5C7432/CP_5C7432 Instance <-> Device 2 (EL6731)/Box 9 (CIM/CIU 150 pump)
//     Standard Inputs/MAIN.HNLT.OuterCapillaryTubeMats.PU600.StatusModule_IN <-> StatusModule/Inputs/StatusModule_0_0
//     Standard Inputs/MAIN.HNLT.OuterCapillaryTubeMats.PU600.fActualSetpoint_IN <-> ActualSetpoint/Inputs/ActualSetpoint_0_0
//     Standard Inputs/MAIN.HNLT.OuterCapillaryTubeMats.PU600.fPowerElectric_IN <-> Power/Inputs/Power_0_0
//     Standard Inputs/MAIN.HNLT.OuterCapillaryTubeMats.PU600.fPowerThermal_IN <-> HeatPower/Inputs/HeatPower_0_0
//     Standard Inputs/MAIN.HNLT.OuterCapillaryTubeMats.PU600.fPressureDifference_IN <-> DiffPressure/Inputs/DiffPressure_0_0
//     Standard Inputs/MAIN.HNLT.OuterCapillaryTubeMats.PU600.fRotationalSpeed_IN <-> Speed/Inputs/Speed_0_0
//     Standard Inputs/MAIN.HNLT.OuterCapillaryTubeMats.PU600.fTemperatureDifference_IN <-> HeatDiffTemp/Inputs/HeatDiffTemp_0_0
//     Standard Inputs/MAIN.HNLT.OuterCapillaryTubeMats.PU600.fTemperatureExternal_IN <-> RemoteTemp2/Inputs/RemoteTemp2_0_0
//     Standard Inputs/MAIN.HNLT.OuterCapillaryTubeMats.PU600.fVolumeFlowRate_IN <-> VolumeFlow/Inputs/VolumeFlow_0_0
//     Standard Inputs/MAIN.HNLT.OuterCapillaryTubeMats.PU600.nAlarmCode_IN <-> FaultCode/Inputs/FaultCode_0_0
//     Standard Inputs/MAIN.HNLT.OuterCapillaryTubeMats.PU600.nWarningCode_IN <-> WarningCode/Inputs/WarningCode_0_0
//     Standard Inputs/MAIN.HNLT.OuterCapillaryTubeMats.PU600.stTemperatureInternal_Genibus_Reply <-> DirectDataReply/Inputs/DirectDataReply_0_0
//     Standard Outputs/MAIN.HNLT.OuterCapillaryTubeMats.PU600.ControlModule_OUT <-> ControlModule/Outputs/ControlModule_1_0
//     Standard Outputs/MAIN.HNLT.OuterCapillaryTubeMats.PU600.stTemperatureInternal_Genibus_Request <-> DirectDataRequest/Outputs/DirectDataRequest_1_0
//   CP_5C7432/CP_5C7432 Instance <-> Device 6 (EL6731)/Box 1 (CIM/CIU 150 pump)
//     Standard Inputs/MAIN.HNHT.AnnealingOvenExhaustGasSystem.PU361.StatusModule_IN <-> StatusModule/Inputs/StatusModule_0_0
//     Standard Inputs/MAIN.HNHT.AnnealingOvenExhaustGasSystem.PU361.fActualSetpoint_IN <-> ActualSetpoint/Inputs/ActualSetpoint_0_0
//     Standard Inputs/MAIN.HNHT.AnnealingOvenExhaustGasSystem.PU361.fPowerElectric_IN <-> Power/Inputs/Power_0_0
//     Standard Inputs/MAIN.HNHT.AnnealingOvenExhaustGasSystem.PU361.fPowerThermal_IN <-> HeatPower/Inputs/HeatPower_0_0
//     Standard Inputs/MAIN.HNHT.AnnealingOvenExhaustGasSystem.PU361.fPressureDifference_IN <-> DiffPressure/Inputs/DiffPressure_0_0
//     Standard Inputs/MAIN.HNHT.AnnealingOvenExhaustGasSystem.PU361.fRotationalSpeed_IN <-> Speed/Inputs/Speed_0_0
//     Standard Inputs/MAIN.HNHT.AnnealingOvenExhaustGasSystem.PU361.fTemperatureDifference_IN <-> HeatDiffTemp/Inputs/HeatDiffTemp_0_0
//     Standard Inputs/MAIN.HNHT.AnnealingOvenExhaustGasSystem.PU361.fTemperatureExternal_IN <-> RemoteTemp2/Inputs/RemoteTemp2_0_0
//     Standard Inputs/MAIN.HNHT.AnnealingOvenExhaustGasSystem.PU361.fVolumeFlowRate_IN <-> VolumeFlow/Inputs/VolumeFlow_0_0
//     Standard Inputs/MAIN.HNHT.AnnealingOvenExhaustGasSystem.PU361.nAlarmCode_IN <-> FaultCode/Inputs/FaultCode_0_0
//     Standard Inputs/MAIN.HNHT.AnnealingOvenExhaustGasSystem.PU361.nWarningCode_IN <-> WarningCode/Inputs/WarningCode_0_0
//     Standard Inputs/MAIN.HNHT.AnnealingOvenExhaustGasSystem.PU361.stTemperatureInternal_Genibus_Reply <-> DirectDataReply/Inputs/DirectDataReply_0_0
//     Standard Outputs/MAIN.HNHT.AnnealingOvenExhaustGasSystem.PU361.ControlModule_OUT <-> ControlModule/Outputs/ControlModule_1_0
//     Standard Outputs/MAIN.HNHT.AnnealingOvenExhaustGasSystem.PU361.stTemperatureInternal_Genibus_Request <-> DirectDataRequest/Outputs/DirectDataRequest_1_0
//   CP_5C7432/CP_5C7432 Instance <-> Device 6 (EL6731)/Box 2 (CIM/CIU 150 pump)
//     Standard Inputs/MAIN.HNLT.AnnealingOvenSealingSystem.PU261.StatusModule_IN <-> StatusModule/Inputs/StatusModule_0_0
//     Standard Inputs/MAIN.HNLT.AnnealingOvenSealingSystem.PU261.fActualSetpoint_IN <-> ActualSetpoint/Inputs/ActualSetpoint_0_0
//     Standard Inputs/MAIN.HNLT.AnnealingOvenSealingSystem.PU261.fPowerElectric_IN <-> Power/Inputs/Power_0_0
//     Standard Inputs/MAIN.HNLT.AnnealingOvenSealingSystem.PU261.fPowerThermal_IN <-> HeatPower/Inputs/HeatPower_0_0
//     Standard Inputs/MAIN.HNLT.AnnealingOvenSealingSystem.PU261.fPressureDifference_IN <-> DiffPressure/Inputs/DiffPressure_0_0
//     Standard Inputs/MAIN.HNLT.AnnealingOvenSealingSystem.PU261.fRotationalSpeed_IN <-> Speed/Inputs/Speed_0_0
//     Standard Inputs/MAIN.HNLT.AnnealingOvenSealingSystem.PU261.fTemperatureDifference_IN <-> HeatDiffTemp/Inputs/HeatDiffTemp_0_0
//     Standard Inputs/MAIN.HNLT.AnnealingOvenSealingSystem.PU261.fTemperatureExternal_IN <-> RemoteTemp2/Inputs/RemoteTemp2_0_0
//     Standard Inputs/MAIN.HNLT.AnnealingOvenSealingSystem.PU261.fVolumeFlowRate_IN <-> VolumeFlow/Inputs/VolumeFlow_0_0
//     Standard Inputs/MAIN.HNLT.AnnealingOvenSealingSystem.PU261.nAlarmCode_IN <-> FaultCode/Inputs/FaultCode_0_0
//     Standard Inputs/MAIN.HNLT.AnnealingOvenSealingSystem.PU261.nWarningCode_IN <-> WarningCode/Inputs/WarningCode_0_0
//     Standard Inputs/MAIN.HNLT.AnnealingOvenSealingSystem.PU261.stTemperatureInternal_Genibus_Reply <-> DirectDataReply/Inputs/DirectDataReply_0_0
//     Standard Outputs/MAIN.HNLT.AnnealingOvenSealingSystem.PU261.ControlModule_OUT <-> ControlModule/Outputs/ControlModule_1_0
//     Standard Outputs/MAIN.HNLT.AnnealingOvenSealingSystem.PU261.stTemperatureInternal_Genibus_Request <-> DirectDataRequest/Outputs/DirectDataRequest_1_0
//   CP_5C7432/CP_5C7432 Instance <-> Device 6 (EL6731)/Box 3 (CIM/CIU 150 pump)
//     Standard Inputs/MAIN.HNHT.CentralMachineHeatingSystem.PU300.StatusModule_IN <-> StatusModule/Inputs/StatusModule_0_0
//     Standard Inputs/MAIN.HNHT.CentralMachineHeatingSystem.PU300.fActualSetpoint_IN <-> ActualSetpoint/Inputs/ActualSetpoint_0_0
//     Standard Inputs/MAIN.HNHT.CentralMachineHeatingSystem.PU300.fPowerElectric_IN <-> Power/Inputs/Power_0_0
//     Standard Inputs/MAIN.HNHT.CentralMachineHeatingSystem.PU300.fPowerThermal_IN <-> HeatPower/Inputs/HeatPower_0_0
//     Standard Inputs/MAIN.HNHT.CentralMachineHeatingSystem.PU300.fPressureDifference_IN <-> DiffPressure/Inputs/DiffPressure_0_0
//     Standard Inputs/MAIN.HNHT.CentralMachineHeatingSystem.PU300.fRotationalSpeed_IN <-> Speed/Inputs/Speed_0_0
//     Standard Inputs/MAIN.HNHT.CentralMachineHeatingSystem.PU300.fTemperatureDifference_IN <-> HeatDiffTemp/Inputs/HeatDiffTemp_0_0
//     Standard Inputs/MAIN.HNHT.CentralMachineHeatingSystem.PU300.fTemperatureExternal_IN <-> RemoteTemp2/Inputs/RemoteTemp2_0_0
//     Standard Inputs/MAIN.HNHT.CentralMachineHeatingSystem.PU300.fVolumeFlowRate_IN <-> VolumeFlow/Inputs/VolumeFlow_0_0
//     Standard Inputs/MAIN.HNHT.CentralMachineHeatingSystem.PU300.nAlarmCode_IN <-> FaultCode/Inputs/FaultCode_0_0
//     Standard Inputs/MAIN.HNHT.CentralMachineHeatingSystem.PU300.nWarningCode_IN <-> WarningCode/Inputs/WarningCode_0_0
//     Standard Inputs/MAIN.HNHT.CentralMachineHeatingSystem.PU300.stTemperatureInternal_Genibus_Reply <-> DirectDataReply/Inputs/DirectDataReply_0_0
//     Standard Outputs/MAIN.HNHT.CentralMachineHeatingSystem.PU300.ControlModule_OUT <-> ControlModule/Outputs/ControlModule_1_0
//     Standard Outputs/MAIN.HNHT.CentralMachineHeatingSystem.PU300.stTemperatureInternal_Genibus_Request <-> DirectDataRequest/Outputs/DirectDataRequest_1_0
//   CP_5C7432/CP_5C7432 Instance <-> Device 6 (EL6731)/Box 4 (CIM/CIU 150 pump)
//     Standard Inputs/MAIN.CN.CentralMachineCoolingSystem.PU100.StatusModule_IN <-> StatusModule/Inputs/StatusModule_0_0
//     Standard Inputs/MAIN.CN.CentralMachineCoolingSystem.PU100.fActualSetpoint_IN <-> ActualSetpoint/Inputs/ActualSetpoint_0_0
//     Standard Inputs/MAIN.CN.CentralMachineCoolingSystem.PU100.fPowerElectric_IN <-> Power/Inputs/Power_0_0
//     Standard Inputs/MAIN.CN.CentralMachineCoolingSystem.PU100.fPowerThermal_IN <-> HeatPower/Inputs/HeatPower_0_0
//     Standard Inputs/MAIN.CN.CentralMachineCoolingSystem.PU100.fPressureDifference_IN <-> DiffPressure/Inputs/DiffPressure_0_0
//     Standard Inputs/MAIN.CN.CentralMachineCoolingSystem.PU100.fRotationalSpeed_IN <-> Speed/Inputs/Speed_0_0
//     Standard Inputs/MAIN.CN.CentralMachineCoolingSystem.PU100.fTemperatureDifference_IN <-> HeatDiffTemp/Inputs/HeatDiffTemp_0_0
//     Standard Inputs/MAIN.CN.CentralMachineCoolingSystem.PU100.fTemperatureExternal_IN <-> RemoteTemp2/Inputs/RemoteTemp2_0_0
//     Standard Inputs/MAIN.CN.CentralMachineCoolingSystem.PU100.fVolumeFlowRate_IN <-> VolumeFlow/Inputs/VolumeFlow_0_0
//     Standard Inputs/MAIN.CN.CentralMachineCoolingSystem.PU100.nAlarmCode_IN <-> FaultCode/Inputs/FaultCode_0_0
//     Standard Inputs/MAIN.CN.CentralMachineCoolingSystem.PU100.nWarningCode_IN <-> WarningCode/Inputs/WarningCode_0_0
//     Standard Inputs/MAIN.CN.CentralMachineCoolingSystem.PU100.stTemperatureInternal_Genibus_Reply <-> DirectDataReply/Inputs/DirectDataReply_0_0
//     Standard Outputs/MAIN.CN.CentralMachineCoolingSystem.PU100.ControlModule_OUT <-> ControlModule/Outputs/ControlModule_1_0
//     Standard Outputs/MAIN.CN.CentralMachineCoolingSystem.PU100.stTemperatureInternal_Genibus_Request <-> DirectDataRequest/Outputs/DirectDataRequest_1_0
//   CP_5C7432/CP_5C7432 Instance <-> Device 6 (EL6731)/Box 6 (CIM/CIU 150 pump)
//     Standard Inputs/MAIN.HNLT.DCSystem.PU245.StatusModule_IN <-> StatusModule/Inputs/StatusModule_0_0
//     Standard Inputs/MAIN.HNLT.DCSystem.PU245.fActualSetpoint_IN <-> ActualSetpoint/Inputs/ActualSetpoint_0_0
//     Standard Inputs/MAIN.HNLT.DCSystem.PU245.fPowerElectric_IN <-> Power/Inputs/Power_0_0
//     Standard Inputs/MAIN.HNLT.DCSystem.PU245.fPowerThermal_IN <-> HeatPower/Inputs/HeatPower_0_0
//     Standard Inputs/MAIN.HNLT.DCSystem.PU245.fPressureDifference_IN <-> DiffPressure/Inputs/DiffPressure_0_0
//     Standard Inputs/MAIN.HNLT.DCSystem.PU245.fRotationalSpeed_IN <-> Speed/Inputs/Speed_0_0
//     Standard Inputs/MAIN.HNLT.DCSystem.PU245.fTemperatureDifference_IN <-> HeatDiffTemp/Inputs/HeatDiffTemp_0_0
//     Standard Inputs/MAIN.HNLT.DCSystem.PU245.fTemperatureExternal_IN <-> RemoteTemp2/Inputs/RemoteTemp2_0_0
//     Standard Inputs/MAIN.HNLT.DCSystem.PU245.fVolumeFlowRate_IN <-> VolumeFlow/Inputs/VolumeFlow_0_0
//     Standard Inputs/MAIN.HNLT.DCSystem.PU245.nAlarmCode_IN <-> FaultCode/Inputs/FaultCode_0_0
//     Standard Inputs/MAIN.HNLT.DCSystem.PU245.nWarningCode_IN <-> WarningCode/Inputs/WarningCode_0_0
//     Standard Inputs/MAIN.HNLT.DCSystem.PU245.stTemperatureInternal_Genibus_Reply <-> DirectDataReply/Inputs/DirectDataReply_0_0
//     Standard Outputs/MAIN.HNLT.DCSystem.PU245.ControlModule_OUT <-> ControlModule/Outputs/ControlModule_1_0
//     Standard Outputs/MAIN.HNLT.DCSystem.PU245.stTemperatureInternal_Genibus_Request <-> DirectDataRequest/Outputs/DirectDataRequest_1_0
//   CP_5C7432/CP_5C7432 Instance <-> Device 7 (OPC UA Virtual)/Client #1
//     Standard Inputs/MAIN.CN.EMAG_Y.ConnectionStatus_IN <-> Inputs/Status/Connected
//   CP_5C7432/CP_5C7432 Instance <-> Device 7 (OPC UA Virtual)/Client #2
//     Standard Inputs/MAIN.HNHT.BvL_CleaningSystem.ConnectionStatus_OPC_BvL <-> Inputs/Status/Connected
//   CP_5C7432/CP_5C7432 Instance <-> Device 7 (OPC UA Virtual)/Client #2/PLC1.MAIN.VarPOU_LoTuS.LoTuS.DAK.BvL_Tanks.BvL_Tank_RZ.Tankheizung.Technische_Waerme.BvL_PWT_UWP_Sek.controlState.bStatusOn
//     Standard Inputs/MAIN.HNHT.BvL_CleaningSystem.Technical_Heat_RZ_UWP <-> Inputs/Value
//   CP_5C7432/CP_5C7432 Instance <-> Device 7 (OPC UA Virtual)/Client #2/PLC1.MAIN.VarPOU_LoTuS.LoTuS.DAK.BvL_Tanks.BvL_Tank_RZ.Tankheizung.Technische_Waerme.BvL_SV_W.controlState.bStatusOn
//     Standard Inputs/MAIN.HNHT.BvL_CleaningSystem.Technical_Heat_RZ_SV <-> Inputs/Value
//   CP_5C7432/CP_5C7432 Instance <-> Device 7 (OPC UA Virtual)/Client #2/PLC1.MAIN.VarPOU_LoTuS.LoTuS.DAK.BvL_Tanks.BvL_Tank_RZ.Tankheizung.Technische_Waerme.Heiz_Soll_Pww.controlState.bStatusOn
//     Standard Inputs/MAIN.HNHT.BvL_CleaningSystem.Technical_Heat_RZ_PWW <-> Inputs/Value
//   CP_5C7432/CP_5C7432 Instance <-> Device 7 (OPC UA Virtual)/Client #2/PLC1.MAIN.VarPOU_LoTuS.LoTuS.DAK.BvL_Tanks.BvL_Tank_SZ.Tankheizung.Technische_Waerme.BvL_PWT_UWP_Sek.controlState.bStatusOn
//     Standard Inputs/MAIN.HNHT.BvL_CleaningSystem.Technical_Heat_SZ_UWP <-> Inputs/Value
//   CP_5C7432/CP_5C7432 Instance <-> Device 7 (OPC UA Virtual)/Client #2/PLC1.MAIN.VarPOU_LoTuS.LoTuS.DAK.BvL_Tanks.BvL_Tank_SZ.Tankheizung.Technische_Waerme.BvL_SV_W.controlState.bStatusOn
//     Standard Inputs/MAIN.HNHT.BvL_CleaningSystem.Technical_Heat_SZ_SV <-> Inputs/Value
//   CP_5C7432/CP_5C7432 Instance <-> Device 7 (OPC UA Virtual)/Client #2/PLC1.MAIN.VarPOU_LoTuS.LoTuS.DAK.BvL_Tanks.BvL_Tank_SZ.Tankheizung.Technische_Waerme.Heiz_Soll_Pww.controlState.bStatusOn
//     Standard Inputs/MAIN.HNHT.BvL_CleaningSystem.Technical_Heat_SZ_PWW <-> Inputs/Value
//   CP_5C7432/CP_5C7432 Instance <-> Device 8 (EtherCAT)/Term 36 (EK1100)/Term 37 (EL2008)
//     Standard Outputs/MAIN.HNLT.CompressorSystem.SVAir{1..6}.bSetStatusOn_OUT <-> Channel {1..6}/Output  (6 links)

CONFIGURATION CP_5C7432
    RESOURCE PLC ON TwinCAT3
        TASK MBus_WZaehler_Task(INTERVAL := T#6ms, PRIORITY := 6);
        TASK MBus_Zaehler_Task(INTERVAL := T#10ms, PRIORITY := 8);
        TASK Standard(INTERVAL := T#20ms, PRIORITY := 10);
        PROGRAM MBUS_WZaehler WITH MBus_WZaehler_Task : MBUS_WZaehler;
        PROGRAM MBUS_WZaehler2 WITH MBus_WZaehler_Task : MBUS_WZaehler2;
        PROGRAM MBUS_WZaehler_Basement WITH MBus_WZaehler_Task : MBUS_WZaehler_Basement;
        PROGRAM MBUS_Zaehler WITH MBus_Zaehler_Task : MBUS_Zaehler;
        PROGRAM MAIN WITH Standard : MAIN;
    END_RESOURCE
END_CONFIGURATION

// ---- DUTs/01 Actuators/pcmChiller/E_PCMControlMode.TcDUT
{attribute 'qualified_only'}
{attribute 'strict'}
TYPE E_PCMControlMode :
(
	coolingMode := 0, 
	pumpMode := 1
);
END_TYPE

// ---- DUTs/01 Actuators/pcmChiller/ST_pcmChillerDefaultParameters.TcDUT
TYPE ST_pcmChillerDefaultParameters :
STRUCT
	aSetPointLimitsTemperature : ARRAY[1..2] OF REAL := [10,28];
END_STRUCT
END_TYPE

// ---- DUTs/01 Actuators/pcmChiller/ST_pcmChillerState.TcDUT
{attribute 'OPC.UA.DA.StructuredType' := '1'}
TYPE ST_pcmChillerState :
STRUCT
	bError	: BOOL;
	fAmbientTemperature : LREAL;
	fMediumOutletTemperature : LREAL; 
	fCoolingCapacity : DINT; 
	fCoolingEER : LREAL; 
	fFlowValue : LREAL; 
	fFanValue : DINT; 
	fCompressorSpeed : DINT; 
	fEEVValue : LREAL; 
	fEEVPosition : DINT; 
	fInputPower : DINT; 
	fEnvironmentTemperature : LREAL;
END_STRUCT
END_TYPE

// ---- DUTs/02 Sensors/ST_JanitzaState.TcDUT
{attribute 'OPC.UA.DA.StructuredType' := '1'}
TYPE ST_JanitzaState :
STRUCT
	fPower 					: REAL;
	sPowerUnit				: STRING := 'kW';
END_STRUCT
END_TYPE

// ---- DUTs/03 Storages/BufferStorage/ST_BufferStorageState.TcDUT
{attribute 'OPC.UA.DA.StructuredType' := '1'}
TYPE ST_BufferStorageState :
STRUCT
	fUpperTemperature 	: REAL;
	fMidTemperature 	: REAL;
	fLowerTemperature 	: REAL;
END_STRUCT
END_TYPE

// ---- DUTs/03 Storages/PCMStorage/ST_PCMStorageState.TcDUT
TYPE ST_PCMStorageState :
STRUCT
	SOCValuePercentage : REAL; 
	SOCValueAbsolute : REAL; 
	TemperatureSensor : REAL; 
END_STRUCT
END_TYPE

// ---- DUTs/04 Systems/ConsumerSystems/CN/ST_CN_CentralMachineCoolingDefaultParameters.TcDUT
TYPE ST_CN_CentralMachineCoolingDefaultParameters :
STRUCT
	aSetPointLimitsRelativeSpeed : ARRAY[1..2] OF REAL := [0,100];
	aSetPointLimitsTemperatureDifference : ARRAY[1..2] OF REAL := [3,5];
END_STRUCT
END_TYPE

// ---- DUTs/04 Systems/ConsumerSystems/CN/ST_FlywheelMassStorageDefaultParameters.TcDUT
TYPE ST_FlywheelMassStorageDefaultParameters :
STRUCT
	aSetPointLimitsRelativeSpeed : ARRAY[1..2] OF REAL := [0,100];
	aSetPointLimitsTemperatureDifference : ARRAY[1..2] OF REAL := [3,5];
END_STRUCT
END_TYPE

// ---- DUTs/04 Systems/ConsumerSystems/HNHT/ST_AnnealingOvenExhaustGasDefaultParameters.TcDUT
TYPE ST_AnnealingOvenExhaustGasDefaultParameters :
STRUCT
	aSetPointLimitsTemperature : ARRAY[1..2] OF REAL := [0,85];
END_STRUCT
END_TYPE

// ---- DUTs/04 Systems/ConsumerSystems/HNHT/ST_HNHT_CentralMachineHeatingDefaultParameters.TcDUT
TYPE ST_HNHT_CentralMachineHeatingDefaultParameters :
STRUCT
	aSetPointLimitsRelativeSpeed : ARRAY[1..2] OF REAL := [0,100];
	aSetPointLimitsTemperatureDifference : ARRAY[1..2] OF REAL := [5,10];
END_STRUCT
END_TYPE

// ---- DUTs/04 Systems/ConsumerSystems/HNLT/ST_DCSystemDefaultParameters.TcDUT
TYPE ST_DCSystemDefaultParameters :
STRUCT
	aSetPointLimitsRelativeSpeed : ARRAY[1..2] OF REAL := [0,100];
	aSetPointLimitsTemperatureDifference : ARRAY[1..2] OF REAL := [3,5];
END_STRUCT
END_TYPE

// ---- DUTs/04 Systems/CoolingSystems/eChiller/ST_eChillerDefaultParameters.TcDUT
TYPE ST_eChillerDefaultParameters :
STRUCT
	aSetPointLimitsTemperature : ARRAY[1..2] OF REAL := [10,28];
END_STRUCT
END_TYPE

// ---- DUTs/04 Systems/CoolingSystems/eChiller/ST_eChillerState.TcDUT
{attribute 'OPC.UA.DA.StructuredType' := '1'}
TYPE ST_eChillerState :
STRUCT
	bError : BOOL;
	bWarning: BOOL;
END_STRUCT
END_TYPE

// ---- DUTs/04 Systems/HeatingSystems/CHP/E_CHPControlMode.TcDUT
{attribute 'qualified_only'}
{attribute 'strict'}
TYPE E_CHPControlMode :
(
	constantPower := 0, 
	supplyTemperature := 1
);
END_TYPE

// ---- DUTs/04 Systems/HeatingSystems/CHP/ST_CHPDefaultParameters.TcDUT
TYPE ST_CHPDefaultParameters :
STRUCT
	fControllerAmplification : LREAL := 5;
	tControllerIntegralTime : TIME := T#100S;
	tTaskCycleTime	: TIME;
	tCtrlCycleTime	: TIME;
	aSetPointLimitsConstantPower : ARRAY[1..2] OF REAL := [50,100];
	aSetPointLimitsTemperature : ARRAY[1..2] OF REAL := [50,90];
END_STRUCT
END_TYPE

// ---- DUTs/04 Systems/HeatingSystems/CHP/ST_CHPSetParameters.TcDUT
{attribute 'OPC.UA.DA.StructuredType' := '1'}
TYPE ST_CHPSetParameters :
STRUCT
	nControlModeAlgorithm : E_CHPControlMode;
	nControlModeManual : E_CHPControlMode;
END_STRUCT
END_TYPE

// ---- DUTs/04 Systems/HeatingSystems/CHP/ST_CHPState.TcDUT
{attribute 'OPC.UA.DA.StructuredType' := '1'}
TYPE ST_CHPState :
STRUCT
	bError					: BOOL;
	fOperatingTime			: UINT;	//hours
	fTemperatureExhaustGas	: INT; //degreeC
	fTemperatureCoolingWater: INT; //degreeC
	fFeedTemperature		: INT; //degreeC
	fReturnTemperature		: INT; //degreeC
	nNumberOfStarts			: UINT;
	fElectricalPower		: INT; //W
	fRotationalSpeed		: UINT;	//rotations per minute
	fGeneratorVoltage		: INT; //V
	fGridVoltage			: INT; //V
	fGeneratorCurrent		: INT; //A
	fCosPhi					: INT;
	nOperationStatus		: UINT;	// 0: Off // 1: Ready // 2: Start // 3: Operating // 4: Error
END_STRUCT
END_TYPE

// ---- DUTs/04 Systems/HeatingSystems/CondensingBoiler/ST_CondensingBoilerDefaultParameters.TcDUT
TYPE ST_CondensingBoilerDefaultParameters :
STRUCT
	aSetPointLimitsTemperature : ARRAY[1..2] OF REAL := [0,80];
END_STRUCT
END_TYPE

// ---- DUTs/04 Systems/HeatingSystems/CondensingBoiler/ST_CondensingBoilerState.TcDUT
{attribute 'OPC.UA.DA.StructuredType' := '1'}
TYPE ST_CondensingBoilerState :
STRUCT
	bError	: BOOL;
END_STRUCT
END_TYPE

// ---- DUTs/04 Systems/HeatingSystems/HeatPump/ST_HeatPumpDefaultParameters.TcDUT
TYPE ST_HeatPumpDefaultParameters :
STRUCT
	aSetPointLimitsTemperature : ARRAY[1..2] OF REAL := [10,100];
END_STRUCT
END_TYPE

// ---- DUTs/04 Systems/HeatingSystems/HeatPump/ST_HeatPumpState.TcDUT
{attribute 'OPC.UA.DA.StructuredType' := '1'}
TYPE ST_HeatPumpState :
STRUCT
	bError	: BOOL;
END_STRUCT
END_TYPE

// ---- DUTs/04 Systems/LinkageSystems/HeatExchanger1/ST_HeatExchanger1DefaultParameters.TcDUT
TYPE ST_HeatExchanger1DefaultParameters :
STRUCT
	aSetPointLimitsTemperature : ARRAY[1..2] OF REAL := [0,100];
END_STRUCT
END_TYPE

// ---- DUTs/04 Systems/LinkageSystems/InnerCapillaryTubeMats/ST_InnerCapillaryTubeMatsDefaultParameters.TcDUT
TYPE ST_InnerCapillaryTubeMatsDefaultParameters :
STRUCT
	aSetPointLimitsTemperature : ARRAY[1..2] OF REAL := [16,45];
	
	//parameters for characteristic heating and cooling curve
	aLimitsAmbientTemperature: ARRAY[1..2] OF REAL := [-5,20];
	aLimitsFeedTemperature: ARRAY[1..2] OF REAL := [40,15];
END_STRUCT
END_TYPE

// ---- DUTs/04 Systems/LinkageSystems/PCMSystem/E_PCMSystemControlMode.TcDUT
{attribute 'qualified_only'}
{attribute 'strict'}
TYPE E_PCMSystemControlMode :
(
	standby := 0,
	directCooling := 1,
	chargePCMChiller := 2,
	dischargePCMchiller := 3	
);
END_TYPE

// ---- DUTs/04 Systems/LinkageSystems/PCMSystem/ST_PCMSystemSetParameters.TcDUT
TYPE ST_PCMSystemSetParameters :
STRUCT
	nControlModeAlgorithm : E_PCMSystemControlMode;
	nControlModeManual : E_PCMSystemControlMode;
END_STRUCT
END_TYPE

// ---- DUTs/04 Systems/LinkageSystems/Ventilation/ST_VentilationDefaultParameters.TcDUT
TYPE ST_VentilationDefaultParameters :
STRUCT
	aSetPointLimitsTemperature : ARRAY[1..2] OF REAL := [16,45];
END_STRUCT
END_TYPE

// ---- DUTs/04 Systems/LinkageSystems/Ventilation/ST_VentilationSetParameters.TcDUT
{attribute 'OPC.UA.DA.StructuredType' := '1'}
TYPE ST_VentilationSetParameters :
STRUCT
	bHeatingModeAlgorithm : BOOL;
	bHeatingModeManual : BOOL;
END_STRUCT
END_TYPE

// ---- DUTs/04 Systems/LinkageSystems/Ventilation/ST_VentilationState.TcDUT
{attribute 'OPC.UA.DA.StructuredType' := '1'}
TYPE ST_VentilationState :
STRUCT
	bError					: BOOL;
	bStatusOnSeminarRoom	: BOOL; //true, if seminar room is active
	bStatusOnStudentRoom	: BOOL; //true, if student room is active
	bStatusOnProductionHall	: BOOL; //true, if hall is active
	bStatusOnClimateRoom 	: BOOL; //true, if climate room is active
	bStatusOnExperimentalMode : BOOL; // true, if experimental mode is on
END_STRUCT
END_TYPE

// ---- DUTs/04 Systems/StorageSystems/ST_ActiveStorageSystemState.TcDUT
{attribute 'OPC.UA.DA.StructuredType' := '1'}
TYPE ST_ActiveStorageSystemState :
STRUCT
	bLoading : BOOL;
	fHeatFlowRate : REAL; //heat flow rate calculated by pump volume flow rate because heat coutner does not work when flow direction changes
END_STRUCT
END_TYPE

// ---- DUTs/05 Thermal Networks/ST_AmbientState.TcDUT
{attribute 'OPC.UA.DA.StructuredType' := '1'}
TYPE ST_AmbientState :
STRUCT
	fOutsideTemperature : REAL;
	fOutsideTemperature_Container : REAL;
	fOutsideTemperature_Mean : REAL;
	fHallTemperature : REAL;
	fRoomTemperature_Container : REAL;
	fWindSpeed : REAL;
	fDawn : REAL;
	bRain : BOOL;
	sTemperatureUnit : STRING := 'degreeC';
	sDawnUnit : STRING := 'lux';
	sWindSpeedUnit : STRING := 'm/s';
	fTemperatureSeminarRoom : REAL; //degreeC
	fCO2SeminarRoom 		: REAL; //Measured CO2 connection in ppm
	fTemperatureStudentRoom : REAL; //degreeC
	fCO2StudentRoom 		: REAL; //Measured CO2 connection in ppm
END_STRUCT
END_TYPE

// ---- DUTs/05 Thermal Networks/ST_CoolingNetworkControl.TcDUT
TYPE ST_CoolingNetworkControl :
STRUCT
	fFeedTemperature : REAL;
	bAlgorithmPermission : BOOL;
	bSetStatusOn_eChiller : BOOL;
	bSetStatusOn_HVFASystem : BOOL;
	bLoading_HVFASystem : BOOL;
END_STRUCT
END_TYPE

// ---- DUTs/05 Thermal Networks/ST_HeatingNetworkHighTemperatureControl.TcDUT
TYPE ST_HeatingNetworkHighTemperatureControl :
STRUCT
	fFeedTemperature : REAL;
	fTargetTemperature : REAL;
	bAlgorithmPermission : BOOL;
	bSetStatusOn_CHP1 : BOOL;
	bSetStatusOn_CHP2 : BOOL;
	bSetStatusOn_CondensingBoiler : BOOL;
	bSetStatusOn_StaticHeating : BOOL;
	bSetStatusOn_VSIStorage : BOOL;
	bLoading_VSISystem : BOOL;
END_STRUCT
END_TYPE

// ---- DUTs/05 Thermal Networks/ST_HnhtHnltLinkageControl.TcDUT
TYPE ST_HnhtHnltLinkageControl :
STRUCT
	fFeedTemperature_HNLT_Heating : REAL;
	fFeedTemperature_HNLT_Cooling : REAL;	
	fFeedTemperature_HNHT : REAL;
	bAlgorithmPermission_HNHT : BOOL;
	bAlgorithmPermission_HNLT : BOOL;
	bSetStatusOn_HeatExchanger1 : BOOL;
	bSetStatusOn_HeatPump : BOOL;
END_STRUCT
END_TYPE

// ---- DUTs/05 Thermal Networks/ST_HnhtCnLinkageControl.TcDUT
TYPE ST_HnhtCnLinkageControl :
STRUCT	
	bHeatingMode : BOOL;
	bAlgorithmPermission_HNHT : BOOL;
	bAlgorithmPermission_CN : BOOL;
END_STRUCT
END_TYPE

// ---- DUTs/06 Strategy/ST_StrategyDefaultParameters.TcDUT
TYPE ST_StrategyDefaultParameters :
STRUCT
	//target temperatures for building mode
	fTargetTemperature_HNHT_Heating : REAL := 55;
	fTargetTemperature_HNHT_Cooling : REAL := 65;
	fTargetTemperature_HNLT_Cooling : REAL := 46;
	fTargetTemperature_HNLT_Heating : REAL := 40;
	fTargetTemperature_CN : REAL := 15;
	
	//temperature limits for thermal networks in building mode
	aTemperatureLimits_HNHT : ARRAY[1..2] OF REAL := [40,85];
	aTemperatureLimits_HNLT : ARRAY[1..2] OF REAL := [25,55];
	aTemperatureLimits_CN : ARRAY[1..2] OF REAL := [10,25];	

	//target temperatures for production mode
	fTargetTemperature_HNHT_Heating_ProductionMode : REAL := 70;
	fTargetTemperature_HNHT_Cooling_ProductionMode : REAL := 80;
	fTargetTemperature_HNLT_Cooling_ProductionMode : REAL := 40;
	fTargetTemperature_HNLT_Heating_ProductionMode : REAL := 34;
	fTargetTemperature_CN_ProductionMode : REAL := 15;
		
	//temperature for thermal networks in production mode
	aTemperatureLimits_HNHT_ProductionMode : ARRAY[1..2] OF REAL := [45,85];
	aTemperatureLimits_HNLT_ProductionMode : ARRAY[1..2] OF REAL := [10,50];
	aTemperatureLimits_CN_ProductionMode : ARRAY[1..2] OF REAL := [10,25];
	
	//offset between target and feed temperatures
	fOffset_FeedTemperature_HNHT : REAL := 4;
	fOffset_FeedTemperature_HNLT_Heating : REAL := 4;
	fOffset_FeedTemperature_HNLT_Cooling : REAL := 6;
	fOffset_FeedTemperature_CN : REAL := 5;
	
	fTargetTemperature_ProductionHall : REAL := 21; //before 19
END_STRUCT
END_TYPE

// ---- DUTs/06 Strategy/ST_StrategySetParameters.TcDUT
{attribute 'OPC.UA.DA.StructuredType' := '1'}
TYPE ST_StrategySetParameters :
STRUCT
	bProductionModeActivated : BOOL;
END_STRUCT
END_TYPE

// ---- DUTs/06 Strategy/ST_StrategyState.TcDUT
{attribute 'OPC.UA.DA.StructuredType' := '1'}
TYPE ST_StrategyState :
STRUCT
	fTargetTemperature_HNHT_Heating : REAL;
	fTargetTemperature_HNHT_Cooling : REAL;
	fTargetTemperature_HNLT_Cooling : REAL;
	fTargetTemperature_HNLT_Heating : REAL;
	fTargetTemperature_CN : REAL;
	fTargetTemperature_ProductionHall : REAL;
	
	aTemperatureLimits_HNHT : ARRAY[1..2] OF REAL;
	aTemperatureLimits_HNLT : ARRAY[1..2] OF REAL;
	aTemperatureLimits_CN : ARRAY[1..2] OF REAL;
	bAlgorithmPermission_HNHT : BOOL;
	bAlgorithmPermission_HNLT : BOOL;
	bAlgorithmPermission_CN : BOOL;

	bHeatingMode : BOOL;	
	
	fFeedTemperature_HNHT : REAL;
	fFeedTemperature_HNLT_Heating : REAL;
	fFeedTemperature_HNLT_Cooling : REAL;
	fFeedTemperature_CN : REAL;
END_STRUCT
END_TYPE

// ---- DUTs/07 Utilities/ST_OPC_UANode.TcDUT
TYPE ST_OPC_UANode :
STRUCT
	NodeID				: ST_UANodeID;
	NodeHdl				: DWORD;
	SizeOfDataType		: UDINT;
	NodeAddInfo			: ST_UANodeAdditionalInfo;
	TargetVar			: POINTER TO BOOL;
END_STRUCT
END_TYPE

// ---- GVLs/GlobalVariables.TcGVL
{attribute 'qualified_only'}
VAR_GLOBAL
	//cycle times
	tTaskCycleTime_MAIN				: TIME := T#50MS;
	tCtrlCycleTime_MAIN				: TIME := T#5S;
	
	//ip addresses
	sIP_EMAG_GT	: STRING := 'opc.tcp://192.168.116.33:4840';
	sIP_FlywheelMassStorage : STRING := 'opc.tcp://192.168.116.110:4840';
	sIP_MAFAC_Java : STRING := 'opc.tcp://192.168.116.47:4840';
	sIP_BvL_CleaningSystem : STRING := 'opc.tcp://192.168.116.129:4840';
	sIP_Annealing_Oven : STRING := 'opc.tcp://192.168.116.16:4840';
	sIP_DC : STRING := 'opc.tcp://192.168.116.41:4840';
	sIP_AbsorptionChiller : STRING := 'opc.tcp://192.168.116.56:4840'; 
	sIP_ImmersionHeater		: STRING := 'opc.tcp://192.168.115.56:4840';
	sIP_HES		: STRING := 'opc.tcp://192.168.115.71:4840';	
	sIP_CompressionChiller		: STRING := 'opc.tcp://192.168.116.19:4840';
	sIP_EMAG_VLC100	: STRING := 'opc.tcp://192.168.116.24:4840';
	sIP_HydraulicDemonstrator : STRING := 'opc.tcp://192.168.115.176:4840';
	sIP_Ventilation : STRING := '192.168.116.58';
	sIP_CHP1 : STRING := '192.168.116.118';
	sIP_CHP2 : STRING := '192.168.116.119';
	sIP_Emonio_HNHT_HeatPump : STRING := '192.168.116.174';
	sIP_Emonio_CN_HeatPump : STRING := '192.168.116.173';
	sIP_Emonio_eChiller : STRING := '192.168.116.177';
	sIP_Emonio_CondensingBoiler : STRING := '192.168.116.167';
	sIP_Emonio_AnnealingOven : STRING := '192.168.116.184';
	sIP_Janitza_Ventilation : STRING := '192.168.116.60';
	
END_VAR

// ---- GVLs/M_Bus.TcGVL
{attribute 'Tc2GvlVarNames'}
VAR_GLOBAL
	IN_Stromzaehler AT %I* 	: ST_KL6781inData22B;
	OUT_Stromzaehler AT %Q* : ST_KL6781outData22B;
	IN_WZaehler AT %I* 	: ST_KL6781inData22B;
	OUT_WZaehler AT %Q* : ST_KL6781outData22B;
	IN_WZaehler2 AT %I* 	: ST_KL6781inData22B;
	OUT_WZaehler2 AT %Q* : ST_KL6781outData22B;
	IN_WZaehler_Basement AT %I* 	: ST_KL6781inData22B;
	OUT_WZaehler_Basement AT %Q* : ST_KL6781outData22B;
	
